LIN {X 0,Y 236.582,Z 268.091,A -85,B 0,C 180,E1 -19847.962,E2 -19847.962} C_VEL
LIN {X 0,Y 237.174,Z 271.955,A -85,B 0,C 180,E1 -19851.515,E2 -19851.515} C_VEL
LIN {X 0,Y 237.168,Z 273.271,A -85,B 0,C 180,E1 -19852.68,E2 -19852.68} C_VEL
LIN {X 0,Y 236.828,Z 274.344,A -85,B 0,C 180,E1 -19853.588,E2 -19853.588} C_VEL
LIN {X 0,Y 235.899,Z 275.46,A -85,B 0,C 180,E1 -19854.474,E2 -19854.474} C_VEL
LIN {X 0,Y 233.05,Z 277.73,A -85,B 0,C 180,E1 -19856.2,E2 -19856.2} C_VEL
LIN {X 0,Y 230.018,Z 280.043,A -85,B 0,C 180,E1 -19857.965,E2 -19857.965} C_VEL
LIN {X 0,Y 228.529,Z 281.776,A -85,B 0,C 180,E1 -19859.356,E2 -19859.356} C_VEL
LIN {X 0,Y 228.311,Z 282.347,A -85,B 0,C 180,E1 -19859.835,E2 -19859.835} C_VEL
LIN {X 0,Y 228.093,Z 283.329,A -85,B 0,C 180,E1 -19860.667,E2 -19860.667} C_VEL
LIN {X 0,Y 230.544,Z 296.949,A -85,B 0,C 180,E1 -19861.77,E2 -19861.77} C_VEL
LIN {X 0,Y 232.298,Z 310.068,A -85,B 0,C 180,E1 -19863.141,E2 -19863.141} C_VEL
LIN {X 0,Y 233.32,Z 321.823,A -85,B 0,C 180,E1 -19864.647,E2 -19864.647} C_VEL
LIN {X 0,Y 233.838,Z 332.507,A -85,B 0,C 180,E1 -19866.296,E2 -19866.296} C_VEL
LIN {X 0,Y 233.74,Z 339.045,A -85,B 0,C 180,E1 -19867.456,E2 -19867.456} C_VEL
LIN {X 0,Y 231.671,Z 349.675,A -85,B 0,C 180,E1 -19869.58,E2 -19869.58} C_VEL
LIN {X 0,Y 229.872,Z 358.64,A -85,B 0,C 180,E1 -19871.823,E2 -19871.823} C_VEL
LIN {X 0,Y 228.341,Z 366.767,A -85,B 0,C 180,E1 -19874.375,E2 -19874.375} C_VEL
LIN {X 0,Y 227.062,Z 373.529,A -85,B 0,C 180,E1 -19877.031,E2 -19877.031} C_VEL
LIN {X 0,Y 226.239,Z 379.732,A -85,B 0,C 180,E1 -19880.161,E2 -19880.161} C_VEL
LIN {X 0,Y 225.922,Z 383.732,A -85,B 0,C 180,E1 -19882.85,E2 -19882.85} C_VEL
LIN {X 0,Y 225.93,Z 385.778,A -85,B 0,C 180,E1 -19884.644,E2 -19884.644} C_VEL
LIN {X 0,Y 225.893,Z 387.38,A -85,B 0,C 180,E1 -19886.431,E2 -19886.431} C_VEL
LIN {X 0,Y 225.931,Z 388.566,A -85,B 0,C 180,E1 -19888.216,E2 -19888.216} C_VEL
LIN {X 0,Y 225.973,Z 389.31,A -85,B 0,C 180,E1 -19889.998,E2 -19889.998} C_VEL
LIN {X 0,Y 225.893,Z 389.616,A -85,B 0,C 180,E1 -19891.781,E2 -19891.781} C_VEL
LIN {X 0,Y 225.727,Z 389.197,A -85,B 0,C 180,E1 -19894.896,E2 -19894.896} C_VEL
LIN {X 0,Y 225.828,Z 388.167,A -85,B 0,C 180,E1 -19897.149,E2 -19897.149} C_VEL
LIN {X 0,Y 226.44,Z 385.148,A -85,B 0,C 180,E1 -19900.731,E2 -19900.731} C_VEL
LIN {X 0,Y 227.36,Z 381.799,A -85,B 0,C 180,E1 -19903.403,E2 -19903.403} C_VEL
LIN {X 0,Y 228.933,Z 377.423,A -85,B 0,C 180,E1 -19906.037,E2 -19906.037} C_VEL
LIN {X 0,Y 231.289,Z 370.883,A -85,B 0,C 180,E1 -19909.064,E2 -19909.064} C_VEL
LIN {X 0,Y 233.668,Z 363.826,A -85,B 0,C 180,E1 -19911.618,E2 -19911.618} C_VEL
LIN {X 0,Y 236.692,Z 355.088,A -85,B 0,C 180,E1 -19914.094,E2 -19914.094} C_VEL
LIN {X 0,Y 239.624,Z 346.258,A -85,B 0,C 180,E1 -19916.098,E2 -19916.098} C_VEL
LIN {X 0,Y 240.747,Z 338.01,A -85,B 0,C 180,E1 -19917.843,E2 -19917.843} C_VEL
LIN {X 0,Y 241.168,Z 328.351,A -85,B 0,C 180,E1 -19919.694,E2 -19919.694} C_VEL
LIN {X 0,Y 240.657,Z 317.965,A -85,B 0,C 180,E1 -19921.527,E2 -19921.527} C_VEL
LIN {X 0,Y 239.299,Z 308.276,A -85,B 0,C 180,E1 -19923.171,E2 -19923.171} C_VEL
LIN {X 0,Y 236.551,Z 295.925,A -85,B 0,C 180,E1 -19925.187,E2 -19925.187} C_VEL
LIN {X 0,Y 233.987,Z 287.833,A -85,B 0,C 180,E1 -19926.545,E2 -19926.545} C_VEL
LIN {X 0,Y 232.504,Z 283.742,A -85,B 0,C 180,E1 -19927.235,E2 -19927.235} C_VEL
LIN {X 0,Y 231.232,Z 280.621,A -85,B 0,C 180,E1 -19927.789,E2 -19927.789} C_VEL
LIN {X 0,Y 231.06,Z 279.554,A -85,B 0,C 180,E1 -19927.942,E2 -19927.942} C_VEL
LIN {X 0,Y 230.865,Z 277.251,A -85,B 0,C 180,E1 -19930.44,E2 -19930.44} C_VEL
LIN {X 0,Y 230.241,Z 273.767,A -85,B 0,C 180,E1 -19934.59,E2 -19934.59} C_VEL
LIN {X 0,Y 229.813,Z 271.38,A -85,B 0,C 180,E1 -19937.714,E2 -19937.714} C_VEL
LIN {X 0,Y 229.314,Z 268.321,A -85,B 0,C 180,E1 -19942.193,E2 -19942.193} C_VEL
LIN {X 0,Y 228.917,Z 265.854,A -85,B 0,C 180,E1 -19946.45,E2 -19946.45} C_VEL
LIN {X 0,Y 228.589,Z 263.894,A -85,B 0,C 180,E1 -19950.53,E2 -19950.53} C_VEL
LIN {X 0,Y 228.326,Z 262.331,A -85,B 0,C 180,E1 -19954.471,E2 -19954.471} C_VEL
LIN {X 0,Y 228.146,Z 261.159,A -85,B 0,C 180,E1 -19958.303,E2 -19958.303} C_VEL
LIN {X 0,Y 228.044,Z 260.181,A -85,B 0,C 180,E1 -19962.812,E2 -19962.812} C_VEL
LIN {X 0,Y 228.091,Z 260.073,A -85,B 0,C 180,E1 -19967.542,E2 -19967.542} C_VEL
LIN {X 0,Y 228.321,Z 260.045,A -85,B 0,C 180,E1 -19971.144,E2 -19971.144} C_VEL
LIN {X 0,Y 228.353,Z 260.04,A -85,B 0,C 180,E1 -19972.926,E2 -19972.926} C_VEL
LIN {X 0,Y 228.55,Z 260.016,A -85,B 0,C 180,E1 -19978.235,E2 -19978.235} C_VEL
LIN {X 0,Y 228.611,Z 260.556,A -85,B 0,C 180,E1 -19981.759,E2 -19981.759} C_VEL
LIN {X 0,Y 228.635,Z 261.873,A -85,B 0,C 180,E1 -19987.06,E2 -19987.06} C_VEL
LIN {X 0,Y 228.673,Z 262.986,A -85,B 0,C 180,E1 -19990.623,E2 -19990.623} C_VEL
LIN {X 0,Y 228.643,Z 264.459,A -85,B 0,C 180,E1 -19994.573,E2 -19994.573} C_VEL
LIN {X 0,Y 229.76,Z 267.333,A -85,B 0,C 180,E1 -19995.124,E2 -19995.124} C_VEL
LIN {X 0,Y 231.658,Z 269.874,A -85,B 0,C 180,E1 -19995.842,E2 -19995.842} C_VEL
LIN {X 0,Y 233.644,Z 273.431,A -85,B 0,C 180,E1 -19996.696,E2 -19996.696} C_VEL
LIN {X 0,Y 237.42,Z 281.431,A -85,B 0,C 180,E1 -19998.483,E2 -19998.483} C_VEL
LIN {X 0,Y 240.96,Z 290.866,A -85,B 0,C 180,E1 -20000.484,E2 -20000.484} C_VEL
LIN {X 0,Y 243.397,Z 299.783,A -85,B 0,C 180,E1 -20002.367,E2 -20002.367} C_VEL
LIN {X 0,Y 245.117,Z 310.056,A -85,B 0,C 180,E1 -20004.563,E2 -20004.563} C_VEL
LIN {X 0,Y 245.334,Z 313.056,A -85,B 0,C 180,E1 -20005.218,E2 -20005.218} C_VEL
LIN {X 0,Y 242.951,Z 322.016,A -85,B 0,C 180,E1 -20006.862,E2 -20006.862} C_VEL
LIN {X 0,Y 240.35,Z 330.299,A -85,B 0,C 180,E1 -20008.695,E2 -20008.695} C_VEL
LIN {X 0,Y 237.533,Z 338.398,A -85,B 0,C 180,E1 -20010.907,E2 -20010.907} C_VEL
LIN {X 0,Y 234.499,Z 346.25,A -85,B 0,C 180,E1 -20013.621,E2 -20013.621} C_VEL
LIN {X 0,Y 231.903,Z 352.66,A -85,B 0,C 180,E1 -20016.5,E2 -20016.5} C_VEL
LIN {X 0,Y 230.178,Z 356.698,A -85,B 0,C 180,E1 -20018.873,E2 -20018.873} C_VEL
LIN {X 0,Y 228.237,Z 360.993,A -85,B 0,C 180,E1 -20022.355,E2 -20022.355} C_VEL
LIN {X 0,Y 226.997,Z 363.354,A -85,B 0,C 180,E1 -20025.401,E2 -20025.401} C_VEL
LIN {X 0,Y 226.239,Z 364.471,A -85,B 0,C 180,E1 -20028.201,E2 -20028.201} C_VEL
LIN {X 0,Y 225.758,Z 364.552,A -85,B 0,C 180,E1 -20031.495,E2 -20031.495} C_VEL
LIN {X 0,Y 225.655,Z 363.668,A -85,B 0,C 180,E1 -20034.067,E2 -20034.067} C_VEL
LIN {X 0,Y 225.915,Z 361.541,A -85,B 0,C 180,E1 -20037.128,E2 -20037.128} C_VEL
LIN {X 0,Y 226.555,Z 358.042,A -85,B 0,C 180,E1 -20040.289,E2 -20040.289} C_VEL
LIN {X 0,Y 227.494,Z 352.709,A -85,B 0,C 180,E1 -20043.616,E2 -20043.616} C_VEL
LIN {X 0,Y 228.704,Z 346.677,A -85,B 0,C 180,E1 -20046.456,E2 -20046.456} C_VEL
LIN {X 0,Y 230.139,Z 339.915,A -85,B 0,C 180,E1 -20048.974,E2 -20048.974} C_VEL
LIN {X 0,Y 231.82,Z 331.64,A -85,B 0,C 180,E1 -20051.44,E2 -20051.44} C_VEL
LIN {X 0,Y 233.769,Z 322.282,A -85,B 0,C 180,E1 -20053.677,E2 -20053.677} C_VEL
LIN {X 0,Y 235.788,Z 311.376,A -85,B 0,C 180,E1 -20055.767,E2 -20055.767} C_VEL
LIN {X 0,Y 237.189,Z 302.379,A -85,B 0,C 180,E1 -20057.162,E2 -20057.162} C_VEL
LIN {X 0,Y 235.414,Z 291.626,A -85,B 0,C 180,E1 -20058.813,E2 -20058.813} C_VEL
LIN {X 0,Y 232.759,Z 279.44,A -85,B 0,C 180,E1 -20060.4,E2 -20060.4} C_VEL
LIN {X 0,Y 229.192,Z 266.831,A -85,B 0,C 180,E1 -20061.788,E2 -20061.788} C_VEL
LIN {X 0,Y 227.359,Z 260.437,A -85,B 0,C 180,E1 -20062.392,E2 -20062.392} C_VEL
LIN {X 0,Y 227.394,Z 260.162,A -85,B 0,C 180,E1 -20062.9,E2 -20062.9} C_VEL
LIN {X 0,Y 227.807,Z 260.108,A -85,B 0,C 180,E1 -20066.464,E2 -20066.464} C_VEL
LIN {X 0,Y 228.552,Z 260.014,A -85,B 0,C 180,E1 -20070.002,E2 -20070.002} C_VEL
LIN {X 0,Y 228.543,Z 260.017,A -85,B 0,C 180,E1 -20071.764,E2 -20071.764} C_VEL
LIN {X 0,Y 228.343,Z 260.043,A -85,B 0,C 180,E1 -20077.074,E2 -20077.074} C_VEL
LIN {X 0,Y 228.152,Z 260.064,A -85,B 0,C 180,E1 -20080.653,E2 -20080.653} C_VEL
LIN {X 0,Y 228.055,Z 260.077,A -85,B 0,C 180,E1 -20086.104,E2 -20086.104} C_VEL
LIN {X 0,Y 227.955,Z 260.089,A -85,B 0,C 180,E1 -20089.826,E2 -20089.826} C_VEL
LIN {X 0,Y 227.92,Z 260.094,A -85,B 0,C 180,E1 -20093.634,E2 -20093.634} C_VEL
LIN {X 0,Y 227.878,Z 260.1,A -85,B 0,C 180,E1 -20097.558,E2 -20097.558} C_VEL
LIN {X 0,Y 227.866,Z 260.102,A -85,B 0,C 180,E1 -20101.625,E2 -20101.625} C_VEL
LIN {X 0,Y 227.895,Z 260.097,A -85,B 0,C 180,E1 -20105.871,E2 -20105.871} C_VEL
LIN {X 0,Y 227.887,Z 260.097,A -85,B 0,C 180,E1 -20110.366,E2 -20110.366} C_VEL
LIN {X 0,Y 227.905,Z 260.097,A -85,B 0,C 180,E1 -20112.723,E2 -20112.723} C_VEL
LIN {X 0,Y 227.895,Z 260.095,A -85,B 0,C 180,E1 -20117.745,E2 -20117.745} C_VEL
LIN {X 0,Y 227.869,Z 260.097,A -85,B 0,C 180,E1 -20121.918,E2 -20121.918} C_VEL
LIN {X 0,Y 227.889,Z 260.084,A -85,B 0,C 180,E1 -20126.377,E2 -20126.377} C_VEL
LIN {X 0,Y 227.918,Z 260.094,A -85,B 0,C 180,E1 -20130.441,E2 -20130.441} C_VEL
LIN {X 0,Y 227.93,Z 260.091,A -85,B 0,C 180,E1 -20134.429,E2 -20134.429} C_VEL
LIN {X 0,Y 227.965,Z 260.076,A -85,B 0,C 180,E1 -20138.291,E2 -20138.291} C_VEL
LIN {X 0,Y 228.039,Z 260.072,A -85,B 0,C 180,E1 -20142.829,E2 -20142.829} C_VEL
LIN {X 0,Y 228.097,Z 260.071,A -85,B 0,C 180,E1 -20147.548,E2 -20147.548} C_VEL
LIN {X 0,Y 228.269,Z 260.044,A -85,B 0,C 180,E1 -20151.147,E2 -20151.147} C_VEL
LIN {X 0,Y 228.324,Z 260.031,A -85,B 0,C 180,E1 -20152.93,E2 -20152.93} C_VEL
LIN {X 0,Y 228.56,Z 260.012,A -85,B 0,C 180,E1 -20158.241,E2 -20158.241} C_VEL
LIN {X 0,Y 228.56,Z 260.016,A -85,B 0,C 180,E1 -20161.765,E2 -20161.765} C_VEL
LIN {X 0,Y 228.322,Z 260.033,A -85,B 0,C 180,E1 -20167.075,E2 -20167.075} C_VEL
LIN {X 0,Y 228.154,Z 260.06,A -85,B 0,C 180,E1 -20170.653,E2 -20170.653} C_VEL
LIN {X 0,Y 228.072,Z 260.074,A -85,B 0,C 180,E1 -20174.274,E2 -20174.274} C_VEL
LIN {X 0,Y 228.014,Z 260.073,A -85,B 0,C 180,E1 -20177.955,E2 -20177.955} C_VEL
LIN {X 0,Y 227.941,Z 260.09,A -85,B 0,C 180,E1 -20182.331,E2 -20182.331} C_VEL
LIN {X 0,Y 227.953,Z 260.086,A -85,B 0,C 180,E1 -20186.604,E2 -20186.604} C_VEL
LIN {X 0,Y 227.908,Z 260.094,A -85,B 0,C 180,E1 -20190.292,E2 -20190.292} C_VEL
LIN {X 0,Y 227.888,Z 260.097,A -85,B 0,C 180,E1 -20193.721,E2 -20193.721} C_VEL
LIN {X 0,Y 227.932,Z 260.16,A -85,B 0,C 180,E1 -20198.668,E2 -20198.668} C_VEL
LIN {X 0,Y 228.56,Z 263.745,A -85,B 0,C 180,E1 -20202.572,E2 -20202.572} C_VEL
LIN {X 0,Y 229.474,Z 268.735,A -85,B 0,C 180,E1 -20207.638,E2 -20207.638} C_VEL
LIN {X 0,Y 230.081,Z 272.478,A -85,B 0,C 180,E1 -20211.228,E2 -20211.228} C_VEL
LIN {X 0,Y 230.054,Z 275.028,A -85,B 0,C 180,E1 -20213.546,E2 -20213.546} C_VEL
LIN {X 0,Y 228.962,Z 279.607,A -85,B 0,C 180,E1 -20217.507,E2 -20217.507} C_VEL
LIN {X 0,Y 228.311,Z 282.347,A -85,B 0,C 180,E1 -20219.835,E2 -20219.835} C_VEL
LIN {X 0,Y 228.247,Z 283.713,A -85,B 0,C 180,E1 -20220.368,E2 -20220.368} C_VEL
LIN {X 0,Y 228.252,Z 286.665,A -85,B 0,C 180,E1 -20220.831,E2 -20220.831} C_VEL
LIN {X 0,Y 227.557,Z 295.044,A -85,B 0,C 180,E1 -20221.333,E2 -20221.333} C_VEL
LIN {X 0,Y 225.695,Z 307.555,A -85,B 0,C 180,E1 -20222.229,E2 -20222.229} C_VEL
LIN {X 0,Y 225.598,Z 311.732,A -85,B 0,C 180,E1 -20222.718,E2 -20222.718} C_VEL
LIN {X 0,Y 226.563,Z 323.939,A -85,B 0,C 180,E1 -20224.408,E2 -20224.408} C_VEL
LIN {X 0,Y 226.931,Z 334.996,A -85,B 0,C 180,E1 -20226.257,E2 -20226.257} C_VEL
LIN {X 0,Y 226.737,Z 340.013,A -85,B 0,C 180,E1 -20227.202,E2 -20227.202} C_VEL
LIN {X 0,Y 224.973,Z 348.459,A -85,B 0,C 180,E1 -20228.944,E2 -20228.944} C_VEL
LIN {X 0,Y 223.066,Z 357.154,A -85,B 0,C 180,E1 -20231.131,E2 -20231.131} C_VEL
LIN {X 0,Y 221.983,Z 363.183,A -85,B 0,C 180,E1 -20232.969,E2 -20232.969} C_VEL
LIN {X 0,Y 220.543,Z 370.59,A -85,B 0,C 180,E1 -20235.7,E2 -20235.7} C_VEL
LIN {X 0,Y 219.632,Z 375.607,A -85,B 0,C 180,E1 -20237.993,E2 -20237.993} C_VEL
LIN {X 0,Y 219.049,Z 380.469,A -85,B 0,C 180,E1 -20240.767,E2 -20240.767} C_VEL
LIN {X 0,Y 218.844,Z 384.179,A -85,B 0,C 180,E1 -20243.544,E2 -20243.544} C_VEL
LIN {X 0,Y 218.815,Z 386.828,A -85,B 0,C 180,E1 -20246.315,E2 -20246.315} C_VEL
LIN {X 0,Y 218.861,Z 388.048,A -85,B 0,C 180,E1 -20248.158,E2 -20248.158} C_VEL
LIN {X 0,Y 218.899,Z 388.852,A -85,B 0,C 180,E1 -20249.998,E2 -20249.998} C_VEL
LIN {X 0,Y 218.819,Z 389.197,A -85,B 0,C 180,E1 -20251.839,E2 -20251.839} C_VEL
LIN {X 0,Y 218.658,Z 388.69,A -85,B 0,C 180,E1 -20255.531,E2 -20255.531} C_VEL
LIN {X 0,Y 218.757,Z 387.862,A -85,B 0,C 180,E1 -20257.381,E2 -20257.381} C_VEL
LIN {X 0,Y 218.998,Z 386.61,A -85,B 0,C 180,E1 -20259.232,E2 -20259.232} C_VEL
LIN {X 0,Y 220.005,Z 382.872,A -85,B 0,C 180,E1 -20262.919,E2 -20262.919} C_VEL
LIN {X 0,Y 221.485,Z 378.926,A -85,B 0,C 180,E1 -20265.645,E2 -20265.645} C_VEL
LIN {X 0,Y 223.37,Z 373.893,A -85,B 0,C 180,E1 -20268.337,E2 -20268.337} C_VEL
LIN {X 0,Y 225.873,Z 367.269,A -85,B 0,C 180,E1 -20271.124,E2 -20271.124} C_VEL
LIN {X 0,Y 228.568,Z 359.988,A -85,B 0,C 180,E1 -20273.559,E2 -20273.559} C_VEL
LIN {X 0,Y 232.041,Z 350.477,A -85,B 0,C 180,E1 -20276.049,E2 -20276.049} C_VEL
LIN {X 0,Y 233.674,Z 344.927,A -85,B 0,C 180,E1 -20277.299,E2 -20277.299} C_VEL
LIN {X 0,Y 234.841,Z 334.364,A -85,B 0,C 180,E1 -20279.568,E2 -20279.568} C_VEL
LIN {X 0,Y 234.903,Z 324.058,A -85,B 0,C 180,E1 -20281.578,E2 -20281.578} C_VEL
LIN {X 0,Y 233.981,Z 313.378,A -85,B 0,C 180,E1 -20283.535,E2 -20283.535} C_VEL
LIN {X 0,Y 231.901,Z 302.017,A -85,B 0,C 180,E1 -20285.546,E2 -20285.546} C_VEL
LIN {X 0,Y 229.361,Z 292.372,A -85,B 0,C 180,E1 -20287.273,E2 -20287.273} C_VEL
LIN {X 0,Y 227.435,Z 286.944,A -85,B 0,C 180,E1 -20288.297,E2 -20288.297} C_VEL
LIN {X 0,Y 226.256,Z 284.042,A -85,B 0,C 180,E1 -20288.857,E2 -20288.857} C_VEL
LIN {X 0,Y 224.405,Z 280.75,A -85,B 0,C 180,E1 -20289.658,E2 -20289.658} C_VEL
LIN {X 0,Y 223.937,Z 278.935,A -85,B 0,C 180,E1 -20289.96,E2 -20289.96} C_VEL
LIN {X 0,Y 223.376,Z 275.767,A -85,B 0,C 180,E1 -20293.8,E2 -20293.8} C_VEL
LIN {X 0,Y 222.755,Z 272.287,A -85,B 0,C 180,E1 -20298.502,E2 -20298.502} C_VEL
LIN {X 0,Y 222.291,Z 269.349,A -85,B 0,C 180,E1 -20303.076,E2 -20303.076} C_VEL
LIN {X 0,Y 221.88,Z 267.008,A -85,B 0,C 180,E1 -20307.418,E2 -20307.418} C_VEL
LIN {X 0,Y 221.586,Z 265.096,A -85,B 0,C 180,E1 -20311.589,E2 -20311.589} C_VEL
LIN {X 0,Y 221.346,Z 263.637,A -85,B 0,C 180,E1 -20315.619,E2 -20315.619} C_VEL
LIN {X 0,Y 221.178,Z 262.571,A -85,B 0,C 180,E1 -20319.539,E2 -20319.539} C_VEL
LIN {X 0,Y 221.152,Z 261.793,A -85,B 0,C 180,E1 -20323.378,E2 -20323.378} C_VEL
LIN {X 0,Y 221.144,Z 261.239,A -85,B 0,C 180,E1 -20329.005,E2 -20329.005} C_VEL
LIN {X 0,Y 221.328,Z 261.175,A -85,B 0,C 180,E1 -20332.7,E2 -20332.7} C_VEL
LIN {X 0,Y 221.614,Z 261.562,A -85,B 0,C 180,E1 -20338.18,E2 -20338.18} C_VEL
LIN {X 0,Y 221.745,Z 261.799,A -85,B 0,C 180,E1 -20339.997,E2 -20339.997} C_VEL
LIN {X 0,Y 221.511,Z 262.564,A -85,B 0,C 180,E1 -20343.635,E2 -20343.635} C_VEL
LIN {X 0,Y 221.7,Z 263.426,A -85,B 0,C 180,E1 -20347.282,E2 -20347.282} C_VEL
LIN {X 0,Y 221.655,Z 264.878,A -85,B 0,C 180,E1 -20351.891,E2 -20351.891} C_VEL
LIN {X 0,Y 221.7,Z 265.259,A -85,B 0,C 180,E1 -20352.527,E2 -20352.527} C_VEL
LIN {X 0,Y 222.844,Z 268.053,A -85,B 0,C 180,E1 -20353.135,E2 -20353.135} C_VEL
LIN {X 0,Y 224.868,Z 270.638,A -85,B 0,C 180,E1 -20353.989,E2 -20353.989} C_VEL
LIN {X 0,Y 226.934,Z 274.226,A -85,B 0,C 180,E1 -20354.972,E2 -20354.972} C_VEL
LIN {X 0,Y 231.406,Z 283.228,A -85,B 0,C 180,E1 -20357.221,E2 -20357.221} C_VEL
LIN {X 0,Y 234.702,Z 291.81,A -85,B 0,C 180,E1 -20359.229,E2 -20359.229} C_VEL
LIN {X 0,Y 237.218,Z 300.932,A -85,B 0,C 180,E1 -20361.277,E2 -20361.277} C_VEL
LIN {X 0,Y 238.783,Z 310.302,A -85,B 0,C 180,E1 -20363.414,E2 -20363.414} C_VEL
LIN {X 0,Y 239.148,Z 314.984,A -85,B 0,C 180,E1 -20364.499,E2 -20364.499} C_VEL
LIN {X 0,Y 235.909,Z 325.925,A -85,B 0,C 180,E1 -20366.658,E2 -20366.658} C_VEL
LIN {X 0,Y 232.762,Z 334.933,A -85,B 0,C 180,E1 -20368.885,E2 -20368.885} C_VEL
LIN {X 0,Y 229.807,Z 342.679,A -85,B 0,C 180,E1 -20371.322,E2 -20371.322} C_VEL
LIN {X 0,Y 226.581,Z 350.194,A -85,B 0,C 180,E1 -20374.345,E2 -20374.345} C_VEL
LIN {X 0,Y 224.11,Z 355.72,A -85,B 0,C 180,E1 -20377.304,E2 -20377.304} C_VEL
LIN {X 0,Y 222.062,Z 360.132,A -85,B 0,C 180,E1 -20380.577,E2 -20380.577} C_VEL
LIN {X 0,Y 220.85,Z 362.435,A -85,B 0,C 180,E1 -20382.955,E2 -20382.955} C_VEL
LIN {X 0,Y 219.917,Z 363.987,A -85,B 0,C 180,E1 -20385.329,E2 -20385.329} C_VEL
LIN {X 0,Y 219.263,Z 364.857,A -85,B 0,C 180,E1 -20387.695,E2 -20387.695} C_VEL
LIN {X 0,Y 218.757,Z 365.07,A -85,B 0,C 180,E1 -20390.443,E2 -20390.443} C_VEL
LIN {X 0,Y 218.581,Z 364.271,A -85,B 0,C 180,E1 -20393.491,E2 -20393.491} C_VEL
LIN {X 0,Y 218.781,Z 362.082,A -85,B 0,C 180,E1 -20396.903,E2 -20396.903} C_VEL
LIN {X 0,Y 219.367,Z 358.998,A -85,B 0,C 180,E1 -20399.877,E2 -20399.877} C_VEL
LIN {X 0,Y 220.269,Z 353.967,A -85,B 0,C 180,E1 -20403.293,E2 -20403.293} C_VEL
LIN {X 0,Y 221.481,Z 348.036,A -85,B 0,C 180,E1 -20406.272,E2 -20406.272} C_VEL
LIN {X 0,Y 223.163,Z 340.423,A -85,B 0,C 180,E1 -20409.252,E2 -20409.252} C_VEL
LIN {X 0,Y 224.875,Z 332.191,A -85,B 0,C 180,E1 -20411.79,E2 -20411.79} C_VEL
LIN {X 0,Y 226.732,Z 323.661,A -85,B 0,C 180,E1 -20413.913,E2 -20413.913} C_VEL
LIN {X 0,Y 228.736,Z 313.328,A -85,B 0,C 180,E1 -20416,E2 -20416} C_VEL
LIN {X 0,Y 230.335,Z 303.125,A -85,B 0,C 180,E1 -20417.669,E2 -20417.669} C_VEL
LIN {X 0,Y 228.601,Z 292.522,A -85,B 0,C 180,E1 -20419.372,E2 -20419.372} C_VEL
LIN {X 0,Y 226.174,Z 281.326,A -85,B 0,C 180,E1 -20420.899,E2 -20420.899} C_VEL
LIN {X 0,Y 222.52,Z 268.016,A -85,B 0,C 180,E1 -20422.433,E2 -20422.433} C_VEL
LIN {X 0,Y 220.395,Z 261.032,A -85,B 0,C 180,E1 -20423.134,E2 -20423.134} C_VEL
LIN {X 0,Y 221.15,Z 260.936,A -85,B 0,C 180,E1 -20428.181,E2 -20428.181} C_VEL
LIN {X 0,Y 221.511,Z 260.891,A -85,B 0,C 180,E1 -20430.002,E2 -20430.002} C_VEL
LIN {X 0,Y 221.501,Z 260.894,A -85,B 0,C 180,E1 -20431.82,E2 -20431.82} C_VEL
LIN {X 0,Y 221.278,Z 260.922,A -85,B 0,C 180,E1 -20437.301,E2 -20437.301} C_VEL
LIN {X 0,Y 221.101,Z 260.944,A -85,B 0,C 180,E1 -20440.997,E2 -20440.997} C_VEL
LIN {X 0,Y 221.015,Z 260.955,A -85,B 0,C 180,E1 -20446.632,E2 -20446.632} C_VEL
LIN {X 0,Y 220.911,Z 260.968,A -85,B 0,C 180,E1 -20450.486,E2 -20450.486} C_VEL
LIN {X 0,Y 220.866,Z 260.974,A -85,B 0,C 180,E1 -20454.437,E2 -20454.437} C_VEL
LIN {X 0,Y 220.829,Z 260.98,A -85,B 0,C 180,E1 -20458.517,E2 -20458.517} C_VEL
LIN {X 0,Y 220.817,Z 260.981,A -85,B 0,C 180,E1 -20462.758,E2 -20462.758} C_VEL
LIN {X 0,Y 220.833,Z 260.977,A -85,B 0,C 180,E1 -20467.291,E2 -20467.291} C_VEL
LIN {X 0,Y 220.849,Z 260.974,A -85,B 0,C 180,E1 -20471.936,E2 -20471.936} C_VEL
LIN {X 0,Y 220.858,Z 260.973,A -85,B 0,C 180,E1 -20477.048,E2 -20477.048} C_VEL
LIN {X 0,Y 220.849,Z 260.974,A -85,B 0,C 180,E1 -20480.477,E2 -20480.477} C_VEL
LIN {X 0,Y 220.814,Z 260.961,A -85,B 0,C 180,E1 -20485.052,E2 -20485.052} C_VEL
LIN {X 0,Y 220.868,Z 260.967,A -85,B 0,C 180,E1 -20489.399,E2 -20489.399} C_VEL
LIN {X 0,Y 220.896,Z 260.967,A -85,B 0,C 180,E1 -20493.553,E2 -20493.553} C_VEL
LIN {X 0,Y 220.88,Z 260.962,A -85,B 0,C 180,E1 -20497.557,E2 -20497.557} C_VEL
LIN {X 0,Y 220.988,Z 260.951,A -85,B 0,C 180,E1 -20502.575,E2 -20502.575} C_VEL
LIN {X 0,Y 221.03,Z 260.95,A -85,B 0,C 180,E1 -20507.143,E2 -20507.143} C_VEL
LIN {X 0,Y 221.207,Z 260.923,A -85,B 0,C 180,E1 -20510.862,E2 -20510.862} C_VEL
LIN {X 0,Y 221.26,Z 260.911,A -85,B 0,C 180,E1 -20512.704,E2 -20512.704} C_VEL
LIN {X 0,Y 221.518,Z 260.889,A -85,B 0,C 180,E1 -20518.185,E2 -20518.185} C_VEL
LIN {X 0,Y 221.517,Z 260.893,A -85,B 0,C 180,E1 -20521.821,E2 -20521.821} C_VEL
LIN {X 0,Y 221.258,Z 260.912,A -85,B 0,C 180,E1 -20527.302,E2 -20527.302} C_VEL
LIN {X 0,Y 221.075,Z 260.943,A -85,B 0,C 180,E1 -20530.999,E2 -20530.999} C_VEL
LIN {X 0,Y 221.027,Z 260.949,A -85,B 0,C 180,E1 -20536.632,E2 -20536.632} C_VEL
LIN {X 0,Y 220.903,Z 260.963,A -85,B 0,C 180,E1 -20540.488,E2 -20540.488} C_VEL
LIN {X 0,Y 220.878,Z 260.97,A -85,B 0,C 180,E1 -20544.436,E2 -20544.436} C_VEL
LIN {X 0,Y 220.838,Z 260.97,A -85,B 0,C 180,E1 -20548.516,E2 -20548.516} C_VEL
LIN {X 0,Y 220.827,Z 260.978,A -85,B 0,C 180,E1 -20552.757,E2 -20552.757} C_VEL
LIN {X 0,Y 220.849,Z 260.974,A -85,B 0,C 180,E1 -20557.779,E2 -20557.779} C_VEL
LIN {X 0,Y 220.856,Z 261.088,A -85,B 0,C 180,E1 -20558.356,E2 -20558.356} C_VEL
LIN {X 0,Y 221.422,Z 264.152,A -85,B 0,C 180,E1 -20561.804,E2 -20561.804} C_VEL
LIN {X 0,Y 222.239,Z 268.736,A -85,B 0,C 180,E1 -20566.667,E2 -20566.667} C_VEL
LIN {X 0,Y 222.999,Z 273.012,A -85,B 0,C 180,E1 -20570.924,E2 -20570.924} C_VEL
LIN {X 0,Y 223.009,Z 275.438,A -85,B 0,C 180,E1 -20573.216,E2 -20573.216} C_VEL
LIN {X 0,Y 222.507,Z 277.787,A -85,B 0,C 180,E1 -20575.349,E2 -20575.349} C_VEL
LIN {X 0,Y 221.196,Z 282.96,A -85,B 0,C 180,E1 -20579.905,E2 -20579.905} C_VEL
LIN {X 0,Y 223.81,Z 297.497,A -85,B 0,C 180,E1 -20581.15,E2 -20581.15} C_VEL
LIN {X 0,Y 225.422,Z 310.201,A -85,B 0,C 180,E1 -20582.532,E2 -20582.532} C_VEL
LIN {X 0,Y 225.598,Z 311.732,A -85,B 0,C 180,E1 -20582.718,E2 -20582.718} C_VEL
LIN {X 0,Y 225.445,Z 317.098,A -85,B 0,C 180,E1 -20583.36,E2 -20583.36} C_VEL
LIN {X 0,Y 223.352,Z 325.814,A -85,B 0,C 180,E1 -20584.431,E2 -20584.431} C_VEL
LIN {X 0,Y 221.242,Z 332.584,A -85,B 0,C 180,E1 -20585.395,E2 -20585.395} C_VEL
LIN {X 0,Y 219.95,Z 339.014,A -85,B 0,C 180,E1 -20586.543,E2 -20586.543} C_VEL
LIN {X 0,Y 218.294,Z 347.241,A -85,B 0,C 180,E1 -20588.267,E2 -20588.267} C_VEL
LIN {X 0,Y 216.457,Z 355.711,A -85,B 0,C 180,E1 -20590.42,E2 -20590.42} C_VEL
LIN {X 0,Y 214.836,Z 363.567,A -85,B 0,C 180,E1 -20592.875,E2 -20592.875} C_VEL
LIN {X 0,Y 213.384,Z 370.834,A -85,B 0,C 180,E1 -20595.697,E2 -20595.697} C_VEL
LIN {X 0,Y 212.38,Z 376.628,A -85,B 0,C 180,E1 -20598.546,E2 -20598.546} C_VEL
LIN {X 0,Y 211.875,Z 381.169,A -85,B 0,C 180,E1 -20601.414,E2 -20601.414} C_VEL
LIN {X 0,Y 211.801,Z 384.857,A -85,B 0,C 180,E1 -20604.563,E2 -20604.563} C_VEL
LIN {X 0,Y 211.791,Z 387.524,A -85,B 0,C 180,E1 -20608.096,E2 -20608.096} C_VEL
LIN {X 0,Y 211.828,Z 388.366,A -85,B 0,C 180,E1 -20609.998,E2 -20609.998} C_VEL
LIN {X 0,Y 211.745,Z 388.775,A -85,B 0,C 180,E1 -20611.9,E2 -20611.9} C_VEL
LIN {X 0,Y 211.576,Z 388.339,A -85,B 0,C 180,E1 -20615.717,E2 -20615.717} C_VEL
LIN {X 0,Y 211.944,Z 386.362,A -85,B 0,C 180,E1 -20619.542,E2 -20619.542} C_VEL
LIN {X 0,Y 213.05,Z 382.706,A -85,B 0,C 180,E1 -20623.349,E2 -20623.349} C_VEL
LIN {X 0,Y 214.631,Z 378.851,A -85,B 0,C 180,E1 -20626.158,E2 -20626.158} C_VEL
LIN {X 0,Y 216.632,Z 373.93,A -85,B 0,C 180,E1 -20628.928,E2 -20628.928} C_VEL
LIN {X 0,Y 219.134,Z 367.697,A -85,B 0,C 180,E1 -20631.689,E2 -20631.689} C_VEL
LIN {X 0,Y 222.081,Z 360.273,A -85,B 0,C 180,E1 -20634.291,E2 -20634.291} C_VEL
LIN {X 0,Y 225.056,Z 352.662,A -85,B 0,C 180,E1 -20636.421,E2 -20636.421} C_VEL
LIN {X 0,Y 226.942,Z 347.404,A -85,B 0,C 180,E1 -20637.677,E2 -20637.677} C_VEL
LIN {X 0,Y 228.177,Z 339.553,A -85,B 0,C 180,E1 -20639.523,E2 -20639.523} C_VEL
LIN {X 0,Y 228.873,Z 330.47,A -85,B 0,C 180,E1 -20641.466,E2 -20641.466} C_VEL
LIN {X 0,Y 228.604,Z 319.825,A -85,B 0,C 180,E1 -20643.597,E2 -20643.597} C_VEL
LIN {X 0,Y 226.92,Z 307.074,A -85,B 0,C 180,E1 -20646.045,E2 -20646.045} C_VEL
LIN {X 0,Y 224.501,Z 296.384,A -85,B 0,C 180,E1 -20648.085,E2 -20648.085} C_VEL
LIN {X 0,Y 222.731,Z 290.929,A -85,B 0,C 180,E1 -20649.196,E2 -20649.196} C_VEL
LIN {X 0,Y 221.699,Z 288.52,A -85,B 0,C 180,E1 -20649.752,E2 -20649.752} C_VEL
LIN {X 0,Y 219.976,Z 284.729,A -85,B 0,C 180,E1 -20650.654,E2 -20650.654} C_VEL
LIN {X 0,Y 217.139,Z 280.2,A -85,B 0,C 180,E1 -20651.98,E2 -20651.98} C_VEL
LIN {X 0,Y 216.583,Z 278.245,A -85,B 0,C 180,E1 -20652.374,E2 -20652.374} C_VEL
LIN {X 0,Y 215.974,Z 274.883,A -85,B 0,C 180,E1 -20656.89,E2 -20656.89} C_VEL
LIN {X 0,Y 215.509,Z 271.708,A -85,B 0,C 180,E1 -20661.709,E2 -20661.709} C_VEL
LIN {X 0,Y 215.032,Z 269.201,A -85,B 0,C 180,E1 -20666.244,E2 -20666.244} C_VEL
LIN {X 0,Y 214.726,Z 267.176,A -85,B 0,C 180,E1 -20670.594,E2 -20670.594} C_VEL
LIN {X 0,Y 214.665,Z 266.308,A -85,B 0,C 180,E1 -20672.716,E2 -20672.716} C_VEL
LIN {X 0,Y 214.409,Z 264.955,A -85,B 0,C 180,E1 -20676.835,E2 -20676.835} C_VEL
LIN {X 0,Y 214.245,Z 263.743,A -85,B 0,C 180,E1 -20682.039,E2 -20682.039} C_VEL
LIN {X 0,Y 214.205,Z 263.107,A -85,B 0,C 180,E1 -20686.72,E2 -20686.72} C_VEL
LIN {X 0,Y 214.381,Z 262.853,A -85,B 0,C 180,E1 -20690.563,E2 -20690.563} C_VEL
LIN {X 0,Y 214.427,Z 262.842,A -85,B 0,C 180,E1 -20692.464,E2 -20692.464} C_VEL
LIN {X 0,Y 214.699,Z 263.175,A -85,B 0,C 180,E1 -20698.121,E2 -20698.121} C_VEL
LIN {X 0,Y 214.845,Z 263.404,A -85,B 0,C 180,E1 -20699.997,E2 -20699.997} C_VEL
LIN {X 0,Y 214.577,Z 264.143,A -85,B 0,C 180,E1 -20703.753,E2 -20703.753} C_VEL
LIN {X 0,Y 214.758,Z 265.017,A -85,B 0,C 180,E1 -20707.519,E2 -20707.519} C_VEL
LIN {X 0,Y 214.77,Z 265.852,A -85,B 0,C 180,E1 -20710.167,E2 -20710.167} C_VEL
LIN {X 0,Y 215.993,Z 268.763,A -85,B 0,C 180,E1 -20710.901,E2 -20710.901} C_VEL
LIN {X 0,Y 218.099,Z 271.443,A -85,B 0,C 180,E1 -20711.91,E2 -20711.91} C_VEL
LIN {X 0,Y 220.107,Z 274.951,A -85,B 0,C 180,E1 -20712.963,E2 -20712.963} C_VEL
LIN {X 0,Y 220.803,Z 275.796,A -85,B 0,C 180,E1 -20713.279,E2 -20713.279} C_VEL
LIN {X 0,Y 224.758,Z 283.509,A -85,B 0,C 180,E1 -20715.469,E2 -20715.469} C_VEL
LIN {X 0,Y 228.547,Z 293.024,A -85,B 0,C 180,E1 -20717.906,E2 -20717.906} C_VEL
LIN {X 0,Y 230.956,Z 301.675,A -85,B 0,C 180,E1 -20720.016,E2 -20720.016} C_VEL
LIN {X 0,Y 232.531,Z 310.694,A -85,B 0,C 180,E1 -20722.194,E2 -20722.194} C_VEL
LIN {X 0,Y 232.998,Z 316.619,A -85,B 0,C 180,E1 -20723.668,E2 -20723.668} C_VEL
LIN {X 0,Y 230.68,Z 324.429,A -85,B 0,C 180,E1 -20725.244,E2 -20725.244} C_VEL
LIN {X 0,Y 227.083,Z 334.308,A -85,B 0,C 180,E1 -20727.657,E2 -20727.657} C_VEL
LIN {X 0,Y 223.918,Z 342.3,A -85,B 0,C 180,E1 -20730.141,E2 -20730.141} C_VEL
LIN {X 0,Y 220.944,Z 348.896,A -85,B 0,C 180,E1 -20732.731,E2 -20732.731} C_VEL
LIN {X 0,Y 218.5,Z 354.151,A -85,B 0,C 180,E1 -20735.374,E2 -20735.374} C_VEL
LIN {X 0,Y 216.031,Z 359.077,A -85,B 0,C 180,E1 -20738.671,E2 -20738.671} C_VEL
LIN {X 0,Y 214.638,Z 361.765,A -85,B 0,C 180,E1 -20741.143,E2 -20741.143} C_VEL
LIN {X 0,Y 213.421,Z 363.798,A -85,B 0,C 180,E1 -20743.747,E2 -20743.747} C_VEL
LIN {X 0,Y 212.383,Z 365.149,A -85,B 0,C 180,E1 -20746.714,E2 -20746.714} C_VEL
LIN {X 0,Y 211.768,Z 365.523,A -85,B 0,C 180,E1 -20749.751,E2 -20749.751} C_VEL
LIN {X 0,Y 211.513,Z 364.689,A -85,B 0,C 180,E1 -20753.269,E2 -20753.269} C_VEL
LIN {X 0,Y 211.598,Z 363.038,A -85,B 0,C 180,E1 -20756.128,E2 -20756.128} C_VEL
LIN {X 0,Y 212.154,Z 359.903,A -85,B 0,C 180,E1 -20759.456,E2 -20759.456} C_VEL
LIN {X 0,Y 213.065,Z 355.148,A -85,B 0,C 180,E1 -20762.941,E2 -20762.941} C_VEL
LIN {X 0,Y 214.095,Z 350.133,A -85,B 0,C 180,E1 -20765.698,E2 -20765.698} C_VEL
LIN {X 0,Y 215.518,Z 343.754,A -85,B 0,C 180,E1 -20768.48,E2 -20768.48} C_VEL
LIN {X 0,Y 217.211,Z 336.143,A -85,B 0,C 180,E1 -20771.124,E2 -20771.124} C_VEL
LIN {X 0,Y 219.17,Z 327.192,A -85,B 0,C 180,E1 -20773.624,E2 -20773.624} C_VEL
LIN {X 0,Y 221.179,Z 317.758,A -85,B 0,C 180,E1 -20775.746,E2 -20775.746} C_VEL
LIN {X 0,Y 223.215,Z 306.722,A -85,B 0,C 180,E1 -20777.731,E2 -20777.731} C_VEL
LIN {X 0,Y 223.449,Z 303.831,A -85,B 0,C 180,E1 -20778.204,E2 -20778.204} C_VEL
LIN {X 0,Y 221.643,Z 292.681,A -85,B 0,C 180,E1 -20780.051,E2 -20780.051} C_VEL
LIN {X 0,Y 219.033,Z 281.045,A -85,B 0,C 180,E1 -20781.7,E2 -20781.7} C_VEL
LIN {X 0,Y 215.422,Z 267.945,A -85,B 0,C 180,E1 -20783.269,E2 -20783.269} C_VEL
LIN {X 0,Y 213.468,Z 261.895,A -85,B 0,C 180,E1 -20783.919,E2 -20783.919} C_VEL
LIN {X 0,Y 214.468,Z 261.769,A -85,B 0,C 180,E1 -20790.002,E2 -20790.002} C_VEL
LIN {X 0,Y 214.434,Z 261.775,A -85,B 0,C 180,E1 -20791.88,E2 -20791.88} C_VEL
LIN {X 0,Y 214.216,Z 261.8,A -85,B 0,C 180,E1 -20797.543,E2 -20797.543} C_VEL
LIN {X 0,Y 214.034,Z 261.826,A -85,B 0,C 180,E1 -20801.364,E2 -20801.364} C_VEL
LIN {X 0,Y 213.927,Z 261.835,A -85,B 0,C 180,E1 -20805.239,E2 -20805.239} C_VEL
LIN {X 0,Y 213.872,Z 261.847,A -85,B 0,C 180,E1 -20809.186,E2 -20809.186} C_VEL
LIN {X 0,Y 213.85,Z 261.846,A -85,B 0,C 180,E1 -20813.229,E2 -20813.229} C_VEL
LIN {X 0,Y 213.821,Z 261.852,A -85,B 0,C 180,E1 -20817.453,E2 -20817.453} C_VEL
LIN {X 0,Y 213.772,Z 261.858,A -85,B 0,C 180,E1 -20821.739,E2 -20821.739} C_VEL
LIN {X 0,Y 213.748,Z 261.861,A -85,B 0,C 180,E1 -20826.29,E2 -20826.29} C_VEL
LIN {X 0,Y 213.789,Z 261.854,A -85,B 0,C 180,E1 -20831.11,E2 -20831.11} C_VEL
LIN {X 0,Y 213.805,Z 261.851,A -85,B 0,C 180,E1 -20833.689,E2 -20833.689} C_VEL
LIN {X 0,Y 213.808,Z 261.849,A -85,B 0,C 180,E1 -20836.352,E2 -20836.352} C_VEL
LIN {X 0,Y 213.777,Z 261.851,A -85,B 0,C 180,E1 -20841.349,E2 -20841.349} C_VEL
LIN {X 0,Y 213.768,Z 261.839,A -85,B 0,C 180,E1 -20846.024,E2 -20846.024} C_VEL
LIN {X 0,Y 213.781,Z 261.855,A -85,B 0,C 180,E1 -20850.458,E2 -20850.458} C_VEL
LIN {X 0,Y 213.803,Z 261.849,A -85,B 0,C 180,E1 -20854.706,E2 -20854.706} C_VEL
LIN {X 0,Y 213.815,Z 261.834,A -85,B 0,C 180,E1 -20858.807,E2 -20858.807} C_VEL
LIN {X 0,Y 213.948,Z 261.827,A -85,B 0,C 180,E1 -20862.807,E2 -20862.807} C_VEL
LIN {X 0,Y 213.985,Z 261.828,A -85,B 0,C 180,E1 -20866.712,E2 -20866.712} C_VEL
LIN {X 0,Y 214.145,Z 261.803,A -85,B 0,C 180,E1 -20870.558,E2 -20870.558} C_VEL
LIN {X 0,Y 214.102,Z 261.798,A -85,B 0,C 180,E1 -20874.352,E2 -20874.352} C_VEL
LIN {X 0,Y 214.451,Z 261.77,A -85,B 0,C 180,E1 -20878.125,E2 -20878.125} C_VEL
LIN {X 0,Y 214.554,Z 261.76,A -85,B 0,C 180,E1 -20880.003,E2 -20880.003} C_VEL
LIN {X 0,Y 214.45,Z 261.772,A -85,B 0,C 180,E1 -20881.881,E2 -20881.881} C_VEL
LIN {X 0,Y 214.199,Z 261.79,A -85,B 0,C 180,E1 -20887.544,E2 -20887.544} C_VEL
LIN {X 0,Y 214.007,Z 261.825,A -85,B 0,C 180,E1 -20891.367,E2 -20891.367} C_VEL
LIN {X 0,Y 213.943,Z 261.836,A -85,B 0,C 180,E1 -20895.239,E2 -20895.239} C_VEL
LIN {X 0,Y 213.85,Z 261.837,A -85,B 0,C 180,E1 -20899.189,E2 -20899.189} C_VEL
LIN {X 0,Y 213.858,Z 261.847,A -85,B 0,C 180,E1 -20903.229,E2 -20903.229} C_VEL
LIN {X 0,Y 213.84,Z 261.842,A -85,B 0,C 180,E1 -20907.451,E2 -20907.451} C_VEL
LIN {X 0,Y 213.779,Z 261.855,A -85,B 0,C 180,E1 -20911.739,E2 -20911.739} C_VEL
LIN {X 0,Y 213.755,Z 261.857,A -85,B 0,C 180,E1 -20916.289,E2 -20916.289} C_VEL
LIN {X 0,Y 213.835,Z 261.919,A -85,B 0,C 180,E1 -20917.924,E2 -20917.924} C_VEL
LIN {X 0,Y 214.479,Z 265.6,A -85,B 0,C 180,E1 -20922.203,E2 -20922.203} C_VEL
LIN {X 0,Y 215.219,Z 269.75,A -85,B 0,C 180,E1 -20926.702,E2 -20926.702} C_VEL
LIN {X 0,Y 215.701,Z 272.268,A -85,B 0,C 180,E1 -20929.332,E2 -20929.332} C_VEL
LIN {X 0,Y 215.972,Z 274.726,A -85,B 0,C 180,E1 -20931.807,E2 -20931.807} C_VEL
LIN {X 0,Y 215.64,Z 277.626,A -85,B 0,C 180,E1 -20934.57,E2 -20934.57} C_VEL
LIN {X 0,Y 214.311,Z 282.601,A -85,B 0,C 180,E1 -20939.122,E2 -20939.122} C_VEL
LIN {X 0,Y 216.768,Z 296.298,A -85,B 0,C 180,E1 -20940.323,E2 -20940.323} C_VEL
LIN {X 0,Y 218.43,Z 308.995,A -85,B 0,C 180,E1 -20941.742,E2 -20941.742} C_VEL
LIN {X 0,Y 219.517,Z 320.87,A -85,B 0,C 180,E1 -20943.368,E2 -20943.368} C_VEL
LIN {X 0,Y 219.982,Z 332.271,A -85,B 0,C 180,E1 -20945.245,E2 -20945.245} C_VEL
LIN {X 0,Y 219.95,Z 339.014,A -85,B 0,C 180,E1 -20946.543,E2 -20946.543} C_VEL
LIN {X 0,Y 219.311,Z 342.138,A -85,B 0,C 180,E1 -20947.155,E2 -20947.155} C_VEL
LIN {X 0,Y 218.046,Z 345.12,A -85,B 0,C 180,E1 -20947.746,E2 -20947.746} C_VEL
LIN {X 0,Y 214.471,Z 350.676,A -85,B 0,C 180,E1 -20948.925,E2 -20948.925} C_VEL
LIN {X 0,Y 209.969,Z 357.192,A -85,B 0,C 180,E1 -20950.576,E2 -20950.576} C_VEL
LIN {X 0,Y 208.439,Z 360.939,A -85,B 0,C 180,E1 -20951.745,E2 -20951.745} C_VEL
LIN {X 0,Y 206.762,Z 368.79,A -85,B 0,C 180,E1 -20954.724,E2 -20954.724} C_VEL
LIN {X 0,Y 205.381,Z 375.809,A -85,B 0,C 180,E1 -20958.15,E2 -20958.15} C_VEL
LIN {X 0,Y 204.841,Z 380.453,A -85,B 0,C 180,E1 -20961.116,E2 -20961.116} C_VEL
LIN {X 0,Y 204.721,Z 384.467,A -85,B 0,C 180,E1 -20964.622,E2 -20964.622} C_VEL
LIN {X 0,Y 204.723,Z 386.991,A -85,B 0,C 180,E1 -20968.031,E2 -20968.031} C_VEL
LIN {X 0,Y 204.758,Z 387.87,A -85,B 0,C 180,E1 -20969.998,E2 -20969.998} C_VEL
LIN {X 0,Y 204.672,Z 388.337,A -85,B 0,C 180,E1 -20971.966,E2 -20971.966} C_VEL
LIN {X 0,Y 204.497,Z 387.987,A -85,B 0,C 180,E1 -20975.916,E2 -20975.916} C_VEL
LIN {X 0,Y 204.909,Z 386.094,A -85,B 0,C 180,E1 -20979.872,E2 -20979.872} C_VEL
LIN {X 0,Y 205.42,Z 384.549,A -85,B 0,C 180,E1 -20981.844,E2 -20981.844} C_VEL
LIN {X 0,Y 206.61,Z 381.449,A -85,B 0,C 180,E1 -20984.779,E2 -20984.779} C_VEL
LIN {X 0,Y 208.475,Z 377.342,A -85,B 0,C 180,E1 -20987.66,E2 -20987.66} C_VEL
LIN {X 0,Y 211.252,Z 371.132,A -85,B 0,C 180,E1 -20990.953,E2 -20990.953} C_VEL
LIN {X 0,Y 213.962,Z 364.447,A -85,B 0,C 180,E1 -20993.725,E2 -20993.725} C_VEL
LIN {X 0,Y 217.477,Z 356.266,A -85,B 0,C 180,E1 -20996.379,E2 -20996.379} C_VEL
LIN {X 0,Y 220.659,Z 348.012,A -85,B 0,C 180,E1 -20998.536,E2 -20998.536} C_VEL
LIN {X 0,Y 222.281,Z 338.373,A -85,B 0,C 180,E1 -21000.896,E2 -21000.896} C_VEL
LIN {X 0,Y 222.849,Z 328.281,A -85,B 0,C 180,E1 -21003.137,E2 -21003.137} C_VEL
LIN {X 0,Y 222.481,Z 318.433,A -85,B 0,C 180,E1 -21005.219,E2 -21005.219} C_VEL
LIN {X 0,Y 220.953,Z 306.676,A -85,B 0,C 180,E1 -21007.609,E2 -21007.609} C_VEL
LIN {X 0,Y 218.405,Z 296.049,A -85,B 0,C 180,E1 -21009.86,E2 -21009.86} C_VEL
LIN {X 0,Y 215.365,Z 288.958,A -85,B 0,C 180,E1 -21011.684,E2 -21011.684} C_VEL
LIN {X 0,Y 213.265,Z 285.211,A -85,B 0,C 180,E1 -21012.833,E2 -21012.833} C_VEL
LIN {X 0,Y 212.468,Z 283.455,A -85,B 0,C 180,E1 -21013.301,E2 -21013.301} C_VEL
LIN {X 0,Y 210.298,Z 280.476,A -85,B 0,C 180,E1 -21014.431,E2 -21014.431} C_VEL
LIN {X 0,Y 209.247,Z 277.536,A -85,B 0,C 180,E1 -21015.14,E2 -21015.14} C_VEL
LIN {X 0,Y 208.934,Z 275.722,A -85,B 0,C 180,E1 -21017.73,E2 -21017.73} C_VEL
LIN {X 0,Y 208.435,Z 272.72,A -85,B 0,C 180,E1 -21022.629,E2 -21022.629} C_VEL
LIN {X 0,Y 208.25,Z 271.436,A -85,B 0,C 180,E1 -21024.987,E2 -21024.987} C_VEL
LIN {X 0,Y 207.884,Z 269.279,A -85,B 0,C 180,E1 -21029.526,E2 -21029.526} C_VEL
LIN {X 0,Y 207.654,Z 267.582,A -85,B 0,C 180,E1 -21033.894,E2 -21033.894} C_VEL
LIN {X 0,Y 207.447,Z 266.324,A -85,B 0,C 180,E1 -21038.117,E2 -21038.117} C_VEL
LIN {X 0,Y 207.358,Z 265.418,A -85,B 0,C 180,E1 -21042.237,E2 -21042.237} C_VEL
LIN {X 0,Y 207.306,Z 264.85,A -85,B 0,C 180,E1 -21046.269,E2 -21046.269} C_VEL
LIN {X 0,Y 207.454,Z 264.55,A -85,B 0,C 180,E1 -21050.245,E2 -21050.245} C_VEL
LIN {X 0,Y 207.536,Z 264.521,A -85,B 0,C 180,E1 -21052.212,E2 -21052.212} C_VEL
LIN {X 0,Y 207.769,Z 264.809,A -85,B 0,C 180,E1 -21058.059,E2 -21058.059} C_VEL
LIN {X 0,Y 207.928,Z 265.002,A -85,B 0,C 180,E1 -21059.997,E2 -21059.997} C_VEL
LIN {X 0,Y 207.662,Z 265.742,A -85,B 0,C 180,E1 -21063.878,E2 -21063.878} C_VEL
LIN {X 0,Y 207.82,Z 266.523,A -85,B 0,C 180,E1 -21067.405,E2 -21067.405} C_VEL
LIN {X 0,Y 209.039,Z 269.479,A -85,B 0,C 180,E1 -21068.273,E2 -21068.273} C_VEL
LIN {X 0,Y 211.483,Z 272.248,A -85,B 0,C 180,E1 -21069.561,E2 -21069.561} C_VEL
LIN {X 0,Y 213.523,Z 275.845,A -85,B 0,C 180,E1 -21070.792,E2 -21070.792} C_VEL
LIN {X 0,Y 214.486,Z 277.366,A -85,B 0,C 180,E1 -21071.335,E2 -21071.335} C_VEL
LIN {X 0,Y 218.657,Z 284.971,A -85,B 0,C 180,E1 -21073.825,E2 -21073.825} C_VEL
LIN {X 0,Y 222.491,Z 294.343,A -85,B 0,C 180,E1 -21076.513,E2 -21076.513} C_VEL
LIN {X 0,Y 224.822,Z 302.604,A -85,B 0,C 180,E1 -21078.685,E2 -21078.685} C_VEL
LIN {X 0,Y 226.444,Z 312.239,A -85,B 0,C 180,E1 -21081.195,E2 -21081.195} C_VEL
LIN {X 0,Y 226.845,Z 319.256,A -85,B 0,C 180,E1 -21083.022,E2 -21083.022} C_VEL
LIN {X 0,Y 223.447,Z 328.875,A -85,B 0,C 180,E1 -21085.102,E2 -21085.102} C_VEL
LIN {X 0,Y 219.982,Z 337.532,A -85,B 0,C 180,E1 -21087.464,E2 -21087.464} C_VEL
LIN {X 0,Y 216.899,Z 344.653,A -85,B 0,C 180,E1 -21089.913,E2 -21089.913} C_VEL
LIN {X 0,Y 213.502,Z 351.591,A -85,B 0,C 180,E1 -21092.927,E2 -21092.927} C_VEL
LIN {X 0,Y 211.233,Z 356.05,A -85,B 0,C 180,E1 -21095.451,E2 -21095.451} C_VEL
LIN {X 0,Y 209.269,Z 359.708,A -85,B 0,C 180,E1 -21098.118,E2 -21098.118} C_VEL
LIN {X 0,Y 207.208,Z 363.239,A -85,B 0,C 180,E1 -21101.742,E2 -21101.742} C_VEL
LIN {X 0,Y 206.086,Z 364.793,A -85,B 0,C 180,E1 -21104.266,E2 -21104.266} C_VEL
LIN {X 0,Y 205.261,Z 365.679,A -85,B 0,C 180,E1 -21106.784,E2 -21106.784} C_VEL
LIN {X 0,Y 204.763,Z 365.937,A -85,B 0,C 180,E1 -21109.3,E2 -21109.3} C_VEL
LIN {X 0,Y 204.441,Z 365.399,A -85,B 0,C 180,E1 -21112.242,E2 -21112.242} C_VEL
LIN {X 0,Y 204.468,Z 363.749,A -85,B 0,C 180,E1 -21115.575,E2 -21115.575} C_VEL
LIN {X 0,Y 204.96,Z 360.758,A -85,B 0,C 180,E1 -21119.049,E2 -21119.049} C_VEL
LIN {X 0,Y 205.851,Z 356.267,A -85,B 0,C 180,E1 -21122.574,E2 -21122.574} C_VEL
LIN {X 0,Y 207.072,Z 350.413,A -85,B 0,C 180,E1 -21125.968,E2 -21125.968} C_VEL
LIN {X 0,Y 208.781,Z 343.001,A -85,B 0,C 180,E1 -21129.222,E2 -21129.222} C_VEL
LIN {X 0,Y 210.655,Z 334.891,A -85,B 0,C 180,E1 -21132.027,E2 -21132.027} C_VEL
LIN {X 0,Y 212.879,Z 325.179,A -85,B 0,C 180,E1 -21134.688,E2 -21134.688} C_VEL
LIN {X 0,Y 215.146,Z 314.331,A -85,B 0,C 180,E1 -21137.029,E2 -21137.029} C_VEL
LIN {X 0,Y 216.618,Z 306.43,A -85,B 0,C 180,E1 -21138.421,E2 -21138.421} C_VEL
LIN {X 0,Y 216.006,Z 300.268,A -85,B 0,C 180,E1 -21139.528,E2 -21139.528} C_VEL
LIN {X 0,Y 213.747,Z 288.194,A -85,B 0,C 180,E1 -21141.494,E2 -21141.494} C_VEL
LIN {X 0,Y 210.449,Z 275.086,A -85,B 0,C 180,E1 -21143.29,E2 -21143.29} C_VEL
LIN {X 0,Y 207.352,Z 265.36,A -85,B 0,C 180,E1 -21144.44,E2 -21144.44} C_VEL
LIN {X 0,Y 206.512,Z 262.762,A -85,B 0,C 180,E1 -21144.754,E2 -21144.754} C_VEL
LIN {X 0,Y 207.424,Z 262.646,A -85,B 0,C 180,E1 -21150.002,E2 -21150.002} C_VEL
LIN {X 0,Y 207.371,Z 262.654,A -85,B 0,C 180,E1 -21151.944,E2 -21151.944} C_VEL
LIN {X 0,Y 207.157,Z 262.678,A -85,B 0,C 180,E1 -21157.801,E2 -21157.801} C_VEL
LIN {X 0,Y 206.971,Z 262.704,A -85,B 0,C 180,E1 -21161.758,E2 -21161.758} C_VEL
LIN {X 0,Y 206.867,Z 262.717,A -85,B 0,C 180,E1 -21165.773,E2 -21165.773} C_VEL
LIN {X 0,Y 206.81,Z 262.724,A -85,B 0,C 180,E1 -21169.868,E2 -21169.868} C_VEL
LIN {X 0,Y 206.761,Z 262.73,A -85,B 0,C 180,E1 -21174.074,E2 -21174.074} C_VEL
LIN {X 0,Y 206.736,Z 262.735,A -85,B 0,C 180,E1 -21178.422,E2 -21178.422} C_VEL
LIN {X 0,Y 206.702,Z 262.737,A -85,B 0,C 180,E1 -21182.959,E2 -21182.959} C_VEL
LIN {X 0,Y 206.72,Z 262.734,A -85,B 0,C 180,E1 -21187.734,E2 -21187.734} C_VEL
LIN {X 0,Y 206.719,Z 262.734,A -85,B 0,C 180,E1 -21191.592,E2 -21191.592} C_VEL
LIN {X 0,Y 206.714,Z 262.73,A -85,B 0,C 180,E1 -21195.562,E2 -21195.562} C_VEL
LIN {X 0,Y 206.718,Z 262.734,A -85,B 0,C 180,E1 -21199.767,E2 -21199.767} C_VEL
LIN {X 0,Y 206.723,Z 262.729,A -85,B 0,C 180,E1 -21202.274,E2 -21202.274} C_VEL
LIN {X 0,Y 206.709,Z 262.724,A -85,B 0,C 180,E1 -21207.048,E2 -21207.048} C_VEL
LIN {X 0,Y 206.768,Z 262.729,A -85,B 0,C 180,E1 -21212.1,E2 -21212.1} C_VEL
LIN {X 0,Y 206.788,Z 262.718,A -85,B 0,C 180,E1 -21216.588,E2 -21216.588} C_VEL
LIN {X 0,Y 206.877,Z 262.704,A -85,B 0,C 180,E1 -21222.2,E2 -21222.2} C_VEL
LIN {X 0,Y 206.918,Z 262.71,A -85,B 0,C 180,E1 -21226.249,E2 -21226.249} C_VEL
LIN {X 0,Y 207.105,Z 262.681,A -85,B 0,C 180,E1 -21230.234,E2 -21230.234} C_VEL
LIN {X 0,Y 207.063,Z 262.674,A -85,B 0,C 180,E1 -21234.159,E2 -21234.159} C_VEL
LIN {X 0,Y 207.388,Z 262.648,A -85,B 0,C 180,E1 -21238.061,E2 -21238.061} C_VEL
LIN {X 0,Y 207.519,Z 262.636,A -85,B 0,C 180,E1 -21240.003,E2 -21240.003} C_VEL
LIN {X 0,Y 207.387,Z 262.652,A -85,B 0,C 180,E1 -21241.945,E2 -21241.945} C_VEL
LIN {X 0,Y 207.142,Z 262.668,A -85,B 0,C 180,E1 -21247.803,E2 -21247.803} C_VEL
LIN {X 0,Y 206.933,Z 262.709,A -85,B 0,C 180,E1 -21251.761,E2 -21251.761} C_VEL
LIN {X 0,Y 206.876,Z 262.713,A -85,B 0,C 180,E1 -21255.773,E2 -21255.773} C_VEL
LIN {X 0,Y 206.795,Z 262.719,A -85,B 0,C 180,E1 -21259.871,E2 -21259.871} C_VEL
LIN {X 0,Y 206.774,Z 262.728,A -85,B 0,C 180,E1 -21264.074,E2 -21264.074} C_VEL
LIN {X 0,Y 206.748,Z 262.725,A -85,B 0,C 180,E1 -21268.421,E2 -21268.421} C_VEL
LIN {X 0,Y 206.71,Z 262.737,A -85,B 0,C 180,E1 -21272.959,E2 -21272.959} C_VEL
LIN {X 0,Y 206.805,Z 262.933,A -85,B 0,C 180,E1 -21277.716,E2 -21277.716} C_VEL
LIN {X 0,Y 207.403,Z 266.333,A -85,B 0,C 180,E1 -21281.797,E2 -21281.797} C_VEL
LIN {X 0,Y 208.134,Z 270.387,A -85,B 0,C 180,E1 -21286.38,E2 -21286.38} C_VEL
LIN {X 0,Y 208.822,Z 274.456,A -85,B 0,C 180,E1 -21290.725,E2 -21290.725} C_VEL
LIN {X 0,Y 208.755,Z 277.619,A -85,B 0,C 180,E1 -21293.904,E2 -21293.904} C_VEL
LIN {X 0,Y 207.43,Z 282.193,A -85,B 0,C 180,E1 -21298.251,E2 -21298.251} C_VEL
LIN {X 0,Y 210.027,Z 296.697,A -85,B 0,C 180,E1 -21299.615,E2 -21299.615} C_VEL
LIN {X 0,Y 211.686,Z 309.637,A -85,B 0,C 180,E1 -21301.144,E2 -21301.144} C_VEL
LIN {X 0,Y 212.738,Z 322.311,A -85,B 0,C 180,E1 -21302.984,E2 -21302.984} C_VEL
LIN {X 0,Y 213.118,Z 334.397,A -85,B 0,C 180,E1 -21305.134,E2 -21305.134} C_VEL
LIN {X 0,Y 212.871,Z 340.63,A -85,B 0,C 180,E1 -21306.4,E2 -21306.4} C_VEL
LIN {X 0,Y 210.836,Z 349.794,A -85,B 0,C 180,E1 -21308.487,E2 -21308.487} C_VEL
LIN {X 0,Y 208.912,Z 358.185,A -85,B 0,C 180,E1 -21310.851,E2 -21310.851} C_VEL
LIN {X 0,Y 208.439,Z 360.939,A -85,B 0,C 180,E1 -21311.745,E2 -21311.745} C_VEL
LIN {X 0,Y 207.035,Z 364.551,A -85,B 0,C 180,E1 -21312.975,E2 -21312.975} C_VEL
LIN {X 0,Y 203.027,Z 369.784,A -85,B 0,C 180,E1 -21315.048,E2 -21315.048} C_VEL
LIN {X 0,Y 199.201,Z 374.315,A -85,B 0,C 180,E1 -21317.326,E2 -21317.326} C_VEL
LIN {X 0,Y 198.114,Z 376.831,A -85,B 0,C 180,E1 -21318.842,E2 -21318.842} C_VEL
LIN {X 0,Y 197.672,Z 381.022,A -85,B 0,C 180,E1 -21321.822,E2 -21321.822} C_VEL
LIN {X 0,Y 197.631,Z 384.104,A -85,B 0,C 180,E1 -21324.719,E2 -21324.719} C_VEL
LIN {X 0,Y 197.657,Z 386.458,A -85,B 0,C 180,E1 -21327.96,E2 -21327.96} C_VEL
LIN {X 0,Y 197.69,Z 387.375,A -85,B 0,C 180,E1 -21329.998,E2 -21329.998} C_VEL
LIN {X 0,Y 197.598,Z 387.878,A -85,B 0,C 180,E1 -21332.036,E2 -21332.036} C_VEL
LIN {X 0,Y 197.412,Z 387.915,A -85,B 0,C 180,E1 -21334.541,E2 -21334.541} C_VEL
LIN {X 0,Y 197.565,Z 386.926,A -85,B 0,C 180,E1 -21338.178,E2 -21338.178} C_VEL
LIN {X 0,Y 198.447,Z 384.352,A -85,B 0,C 180,E1 -21342.266,E2 -21342.266} C_VEL
LIN {X 0,Y 199.727,Z 381.319,A -85,B 0,C 180,E1 -21345.3,E2 -21345.3} C_VEL
LIN {X 0,Y 201.676,Z 377.299,A -85,B 0,C 180,E1 -21348.276,E2 -21348.276} C_VEL
LIN {X 0,Y 204.181,Z 372.214,A -85,B 0,C 180,E1 -21351.185,E2 -21351.185} C_VEL
LIN {X 0,Y 206.968,Z 365.927,A -85,B 0,C 180,E1 -21354.045,E2 -21354.045} C_VEL
LIN {X 0,Y 210.528,Z 358.174,A -85,B 0,C 180,E1 -21356.784,E2 -21356.784} C_VEL
LIN {X 0,Y 213.901,Z 350.353,A -85,B 0,C 180,E1 -21358.986,E2 -21358.986} C_VEL
LIN {X 0,Y 215.198,Z 345.008,A -85,B 0,C 180,E1 -21360.409,E2 -21360.409} C_VEL
LIN {X 0,Y 216.517,Z 336.146,A -85,B 0,C 180,E1 -21362.61,E2 -21362.61} C_VEL
LIN {X 0,Y 216.945,Z 326.407,A -85,B 0,C 180,E1 -21364.876,E2 -21364.876} C_VEL
LIN {X 0,Y 216.321,Z 315.403,A -85,B 0,C 180,E1 -21367.316,E2 -21367.316} C_VEL
LIN {X 0,Y 214.779,Z 304.905,A -85,B 0,C 180,E1 -21369.637,E2 -21369.637} C_VEL
LIN {X 0,Y 213.565,Z 299.896,A -85,B 0,C 180,E1 -21370.806,E2 -21370.806} C_VEL
LIN {X 0,Y 211.453,Z 294.435,A -85,B 0,C 180,E1 -21372.306,E2 -21372.306} C_VEL
LIN {X 0,Y 209.109,Z 289.698,A -85,B 0,C 180,E1 -21373.819,E2 -21373.819} C_VEL
LIN {X 0,Y 206.27,Z 284.798,A -85,B 0,C 180,E1 -21375.57,E2 -21375.57} C_VEL
LIN {X 0,Y 205.529,Z 283.095,A -85,B 0,C 180,E1 -21376.08,E2 -21376.08} C_VEL
LIN {X 0,Y 203.055,Z 279.844,A -85,B 0,C 180,E1 -21377.597,E2 -21377.597} C_VEL
LIN {X 0,Y 201.864,Z 276.646,A -85,B 0,C 180,E1 -21378.583,E2 -21378.583} C_VEL
LIN {X 0,Y 201.453,Z 273.728,A -85,B 0,C 180,E1 -21383.622,E2 -21383.622} C_VEL
LIN {X 0,Y 201.019,Z 271.44,A -85,B 0,C 180,E1 -21388.367,E2 -21388.367} C_VEL
LIN {X 0,Y 200.789,Z 269.606,A -85,B 0,C 180,E1 -21392.93,E2 -21392.93} C_VEL
LIN {X 0,Y 200.563,Z 268.247,A -85,B 0,C 180,E1 -21397.325,E2 -21397.325} C_VEL
LIN {X 0,Y 200.47,Z 267.256,A -85,B 0,C 180,E1 -21401.605,E2 -21401.605} C_VEL
LIN {X 0,Y 200.4,Z 266.63,A -85,B 0,C 180,E1 -21405.786,E2 -21405.786} C_VEL
LIN {X 0,Y 200.535,Z 266.277,A -85,B 0,C 180,E1 -21409.905,E2 -21409.905} C_VEL
LIN {X 0,Y 200.632,Z 266.204,A -85,B 0,C 180,E1 -21411.942,E2 -21411.942} C_VEL
LIN {X 0,Y 200.853,Z 266.436,A -85,B 0,C 180,E1 -21417.992,E2 -21417.992} C_VEL
LIN {X 0,Y 201.038,Z 266.628,A -85,B 0,C 180,E1 -21419.997,E2 -21419.997} C_VEL
LIN {X 0,Y 200.771,Z 267.49,A -85,B 0,C 180,E1 -21424.074,E2 -21424.074} C_VEL
LIN {X 0,Y 201.957,Z 270.238,A -85,B 0,C 180,E1 -21425.05,E2 -21425.05} C_VEL
LIN {X 0,Y 204.791,Z 273.044,A -85,B 0,C 180,E1 -21426.79,E2 -21426.79} C_VEL
LIN {X 0,Y 206.461,Z 276.2,A -85,B 0,C 180,E1 -21428.007,E2 -21428.007} C_VEL
LIN {X 0,Y 207.752,Z 277.575,A -85,B 0,C 180,E1 -21428.753,E2 -21428.753} C_VEL
LIN {X 0,Y 209.752,Z 281.349,A -85,B 0,C 180,E1 -21430.128,E2 -21430.128} C_VEL
LIN {X 0,Y 213.519,Z 288.576,A -85,B 0,C 180,E1 -21432.708,E2 -21432.708} C_VEL
LIN {X 0,Y 216.553,Z 295.951,A -85,B 0,C 180,E1 -21435.045,E2 -21435.045} C_VEL
LIN {X 0,Y 219.026,Z 304.865,A -85,B 0,C 180,E1 -21437.624,E2 -21437.624} C_VEL
LIN {X 0,Y 220.477,Z 313.95,A -85,B 0,C 180,E1 -21440.158,E2 -21440.158} C_VEL
LIN {X 0,Y 220.829,Z 320.376,A -85,B 0,C 180,E1 -21441.963,E2 -21441.963} C_VEL
LIN {X 0,Y 219.307,Z 325.152,A -85,B 0,C 180,E1 -21443.024,E2 -21443.024} C_VEL
LIN {X 0,Y 215.5,Z 334.72,A -85,B 0,C 180,E1 -21445.442,E2 -21445.442} C_VEL
LIN {X 0,Y 212.225,Z 342.043,A -85,B 0,C 180,E1 -21447.764,E2 -21447.764} C_VEL
LIN {X 0,Y 209.131,Z 348.372,A -85,B 0,C 180,E1 -21450.267,E2 -21450.267} C_VEL
LIN {X 0,Y 206.124,Z 353.966,A -85,B 0,C 180,E1 -21453.057,E2 -21453.057} C_VEL
LIN {X 0,Y 203.674,Z 358.353,A -85,B 0,C 180,E1 -21455.912,E2 -21455.912} C_VEL
LIN {X 0,Y 201.13,Z 362.582,A -85,B 0,C 180,E1 -21459.763,E2 -21459.763} C_VEL
LIN {X 0,Y 199.776,Z 364.523,A -85,B 0,C 180,E1 -21462.377,E2 -21462.377} C_VEL
LIN {X 0,Y 198.719,Z 365.737,A -85,B 0,C 180,E1 -21465.013,E2 -21465.013} C_VEL
LIN {X 0,Y 197.842,Z 366.333,A -85,B 0,C 180,E1 -21468.239,E2 -21468.239} C_VEL
LIN {X 0,Y 197.402,Z 365.922,A -85,B 0,C 180,E1 -21471.554,E2 -21471.554} C_VEL
LIN {X 0,Y 197.348,Z 364.242,A -85,B 0,C 180,E1 -21475.267,E2 -21475.267} C_VEL
LIN {X 0,Y 197.751,Z 361.644,A -85,B 0,C 180,E1 -21478.527,E2 -21478.527} C_VEL
LIN {X 0,Y 198.393,Z 358.537,A -85,B 0,C 180,E1 -21481.294,E2 -21481.294} C_VEL
LIN {X 0,Y 199.546,Z 352.988,A -85,B 0,C 180,E1 -21485.001,E2 -21485.001} C_VEL
LIN {X 0,Y 201.168,Z 345.968,A -85,B 0,C 180,E1 -21488.482,E2 -21488.482} C_VEL
LIN {X 0,Y 202.917,Z 338.703,A -85,B 0,C 180,E1 -21491.317,E2 -21491.317} C_VEL
LIN {X 0,Y 205.044,Z 329.797,A -85,B 0,C 180,E1 -21494.088,E2 -21494.088} C_VEL
LIN {X 0,Y 207.431,Z 319.28,A -85,B 0,C 180,E1 -21496.667,E2 -21496.667} C_VEL
LIN {X 0,Y 209.531,Z 308.998,A -85,B 0,C 180,E1 -21498.677,E2 -21498.677} C_VEL
LIN {X 0,Y 209.814,Z 305.692,A -85,B 0,C 180,E1 -21499.262,E2 -21499.262} C_VEL
LIN {X 0,Y 208.065,Z 294.669,A -85,B 0,C 180,E1 -21501.269,E2 -21501.269} C_VEL
LIN {X 0,Y 205.513,Z 283.062,A -85,B 0,C 180,E1 -21503.079,E2 -21503.079} C_VEL
LIN {X 0,Y 202.166,Z 270.85,A -85,B 0,C 180,E1 -21504.704,E2 -21504.704} C_VEL
LIN {X 0,Y 199.534,Z 263.63,A -85,B 0,C 180,E1 -21505.646,E2 -21505.646} C_VEL
LIN {X 0,Y 200.379,Z 263.524,A -85,B 0,C 180,E1 -21510.002,E2 -21510.002} C_VEL
LIN {X 0,Y 200.31,Z 263.534,A -85,B 0,C 180,E1 -21512.013,E2 -21512.013} C_VEL
LIN {X 0,Y 200.1,Z 263.557,A -85,B 0,C 180,E1 -21518.078,E2 -21518.078} C_VEL
LIN {X 0,Y 199.903,Z 263.584,A -85,B 0,C 180,E1 -21522.18,E2 -21522.18} C_VEL
LIN {X 0,Y 199.805,Z 263.596,A -85,B 0,C 180,E1 -21526.346,E2 -21526.346} C_VEL
LIN {X 0,Y 199.739,Z 263.604,A -85,B 0,C 180,E1 -21530.603,E2 -21530.603} C_VEL
LIN {X 0,Y 199.669,Z 263.618,A -85,B 0,C 180,E1 -21534.987,E2 -21534.987} C_VEL
LIN {X 0,Y 199.668,Z 263.615,A -85,B 0,C 180,E1 -21539.526,E2 -21539.526} C_VEL
LIN {X 0,Y 199.658,Z 263.618,A -85,B 0,C 180,E1 -21542.356,E2 -21542.356} C_VEL
LIN {X 0,Y 199.647,Z 263.619,A -85,B 0,C 180,E1 -21546.76,E2 -21546.76} C_VEL
LIN {X 0,Y 199.673,Z 263.609,A -85,B 0,C 180,E1 -21549.315,E2 -21549.315} C_VEL
LIN {X 0,Y 199.658,Z 263.616,A -85,B 0,C 180,E1 -21552.342,E2 -21552.342} C_VEL
LIN {X 0,Y 199.662,Z 263.609,A -85,B 0,C 180,E1 -21555.257,E2 -21555.257} C_VEL
LIN {X 0,Y 199.659,Z 263.614,A -85,B 0,C 180,E1 -21558.03,E2 -21558.03} C_VEL
LIN {X 0,Y 199.677,Z 263.609,A -85,B 0,C 180,E1 -21560.747,E2 -21560.747} C_VEL
LIN {X 0,Y 199.633,Z 263.596,A -85,B 0,C 180,E1 -21565.722,E2 -21565.722} C_VEL
LIN {X 0,Y 199.704,Z 263.598,A -85,B 0,C 180,E1 -21568.142,E2 -21568.142} C_VEL
LIN {X 0,Y 199.688,Z 263.61,A -85,B 0,C 180,E1 -21572.776,E2 -21572.776} C_VEL
LIN {X 0,Y 199.74,Z 263.594,A -85,B 0,C 180,E1 -21577.233,E2 -21577.233} C_VEL
LIN {X 0,Y 199.8,Z 263.582,A -85,B 0,C 180,E1 -21581.761,E2 -21581.761} C_VEL
LIN {X 0,Y 199.853,Z 263.589,A -85,B 0,C 180,E1 -21585.753,E2 -21585.753} C_VEL
LIN {X 0,Y 200.028,Z 263.565,A -85,B 0,C 180,E1 -21589.885,E2 -21589.885} C_VEL
LIN {X 0,Y 200.025,Z 263.549,A -85,B 0,C 180,E1 -21593.953,E2 -21593.953} C_VEL
LIN {X 0,Y 200.327,Z 263.527,A -85,B 0,C 180,E1 -21597.993,E2 -21597.993} C_VEL
LIN {X 0,Y 200.484,Z 263.512,A -85,B 0,C 180,E1 -21600.003,E2 -21600.003} C_VEL
LIN {X 0,Y 200.028,Z 263.564,A -85,B 0,C 180,E1 -21604.033,E2 -21604.033} C_VEL
LIN {X 0,Y 200.092,Z 263.546,A -85,B 0,C 180,E1 -21608.08,E2 -21608.08} C_VEL
LIN {X 0,Y 199.883,Z 263.586,A -85,B 0,C 180,E1 -21612.182,E2 -21612.182} C_VEL
LIN {X 0,Y 199.814,Z 263.591,A -85,B 0,C 180,E1 -21616.346,E2 -21616.346} C_VEL
LIN {X 0,Y 199.711,Z 263.602,A -85,B 0,C 180,E1 -21620.607,E2 -21620.607} C_VEL
LIN {X 0,Y 199.684,Z 263.612,A -85,B 0,C 180,E1 -21624.986,E2 -21624.986} C_VEL
LIN {X 0,Y 199.676,Z 263.611,A -85,B 0,C 180,E1 -21629.525,E2 -21629.525} C_VEL
LIN {X 0,Y 199.682,Z 263.611,A -85,B 0,C 180,E1 -21632.357,E2 -21632.357} C_VEL
LIN {X 0,Y 199.731,Z 263.719,A -85,B 0,C 180,E1 -21637.216,E2 -21637.216} C_VEL
LIN {X 0,Y 200.395,Z 267.391,A -85,B 0,C 180,E1 -21641.789,E2 -21641.789} C_VEL
LIN {X 0,Y 201.23,Z 272.037,A -85,B 0,C 180,E1 -21647.178,E2 -21647.178} C_VEL
LIN {X 0,Y 201.773,Z 275.67,A -85,B 0,C 180,E1 -21651.171,E2 -21651.171} C_VEL
LIN {X 0,Y 201.713,Z 278.098,A -85,B 0,C 180,E1 -21653.677,E2 -21653.677} C_VEL
LIN {X 0,Y 200.598,Z 281.867,A -85,B 0,C 180,E1 -21657.4,E2 -21657.4} C_VEL
LIN {X 0,Y 203.003,Z 295.504,A -85,B 0,C 180,E1 -21658.691,E2 -21658.691} C_VEL
LIN {X 0,Y 204.704,Z 308.099,A -85,B 0,C 180,E1 -21660.215,E2 -21660.215} C_VEL
LIN {X 0,Y 205.704,Z 320.209,A -85,B 0,C 180,E1 -21661.996,E2 -21661.996} C_VEL
LIN {X 0,Y 206.146,Z 331.303,A -85,B 0,C 180,E1 -21663.962,E2 -21663.962} C_VEL
LIN {X 0,Y 206.044,Z 340.281,A -85,B 0,C 180,E1 -21665.836,E2 -21665.836} C_VEL
LIN {X 0,Y 203.701,Z 350.506,A -85,B 0,C 180,E1 -21668.28,E2 -21668.28} C_VEL
LIN {X 0,Y 201.837,Z 358.628,A -85,B 0,C 180,E1 -21670.7,E2 -21670.7} C_VEL
LIN {X 0,Y 200.108,Z 366.671,A -85,B 0,C 180,E1 -21673.68,E2 -21673.68} C_VEL
LIN {X 0,Y 198.71,Z 373.148,A -85,B 0,C 180,E1 -21676.707,E2 -21676.707} C_VEL
LIN {X 0,Y 198.114,Z 376.831,A -85,B 0,C 180,E1 -21678.842,E2 -21678.842} C_VEL
LIN {X 0,Y 197.162,Z 379.152,A -85,B 0,C 180,E1 -21680.401,E2 -21680.401} C_VEL
LIN {X 0,Y 194.033,Z 382.213,A -85,B 0,C 180,E1 -21683.014,E2 -21683.014} C_VEL
LIN {X 0,Y 191.573,Z 384.113,A -85,B 0,C 180,E1 -21685.203,E2 -21685.203} C_VEL
LIN {X 0,Y 190.602,Z 385.318,A -85,B 0,C 180,E1 -21686.927,E2 -21686.927} C_VEL
LIN {X 0,Y 190.559,Z 385.665,A -85,B 0,C 180,E1 -21687.512,E2 -21687.512} C_VEL
LIN {X 0,Y 190.623,Z 386.869,A -85,B 0,C 180,E1 -21689.998,E2 -21689.998} C_VEL
LIN {X 0,Y 190.501,Z 387.41,A -85,B 0,C 180,E1 -21692.112,E2 -21692.112} C_VEL
LIN {X 0,Y 190.337,Z 387.554,A -85,B 0,C 180,E1 -21694.447,E2 -21694.447} C_VEL
LIN {X 0,Y 190.509,Z 386.623,A -85,B 0,C 180,E1 -21698.484,E2 -21698.484} C_VEL
LIN {X 0,Y 191.473,Z 384.132,A -85,B 0,C 180,E1 -21702.72,E2 -21702.72} C_VEL
LIN {X 0,Y 192.867,Z 381.199,A -85,B 0,C 180,E1 -21705.858,E2 -21705.858} C_VEL
LIN {X 0,Y 194.906,Z 377.296,A -85,B 0,C 180,E1 -21708.935,E2 -21708.935} C_VEL
LIN {X 0,Y 197.558,Z 372.324,A -85,B 0,C 180,E1 -21711.931,E2 -21711.931} C_VEL
LIN {X 0,Y 200.496,Z 366.156,A -85,B 0,C 180,E1 -21714.872,E2 -21714.872} C_VEL
LIN {X 0,Y 204.22,Z 358.577,A -85,B 0,C 180,E1 -21717.681,E2 -21717.681} C_VEL
LIN {X 0,Y 207.729,Z 350.944,A -85,B 0,C 180,E1 -21719.933,E2 -21719.933} C_VEL
LIN {X 0,Y 209.81,Z 342.068,A -85,B 0,C 180,E1 -21722.406,E2 -21722.406} C_VEL
LIN {X 0,Y 210.806,Z 333.802,A -85,B 0,C 180,E1 -21724.522,E2 -21724.522} C_VEL
LIN {X 0,Y 211.079,Z 323.762,A -85,B 0,C 180,E1 -21726.953,E2 -21726.953} C_VEL
LIN {X 0,Y 210.443,Z 313.447,A -85,B 0,C 180,E1 -21729.382,E2 -21729.382} C_VEL
LIN {X 0,Y 208.823,Z 304.139,A -85,B 0,C 180,E1 -21731.653,E2 -21731.653} C_VEL
LIN {X 0,Y 207.071,Z 299.245,A -85,B 0,C 180,E1 -21733.133,E2 -21733.133} C_VEL
LIN {X 0,Y 204.976,Z 294.556,A -85,B 0,C 180,E1 -21734.709,E2 -21734.709} C_VEL
LIN {X 0,Y 202.555,Z 289.926,A -85,B 0,C 180,E1 -21736.464,E2 -21736.464} C_VEL
LIN {X 0,Y 201.86,Z 288.572,A -85,B 0,C 180,E1 -21736.979,E2 -21736.979} C_VEL
LIN {X 0,Y 199.671,Z 285.096,A -85,B 0,C 180,E1 -21738.546,E2 -21738.546} C_VEL
LIN {X 0,Y 198.486,Z 282.444,A -85,B 0,C 180,E1 -21739.531,E2 -21739.531} C_VEL
LIN {X 0,Y 195.638,Z 278.729,A -85,B 0,C 180,E1 -21741.704,E2 -21741.704} C_VEL
LIN {X 0,Y 194.555,Z 275.685,A -85,B 0,C 180,E1 -21742.873,E2 -21742.873} C_VEL
LIN {X 0,Y 194.21,Z 273.615,A -85,B 0,C 180,E1 -21747.121,E2 -21747.121} C_VEL
LIN {X 0,Y 193.927,Z 271.648,A -85,B 0,C 180,E1 -21751.889,E2 -21751.889} C_VEL
LIN {X 0,Y 193.696,Z 270.185,A -85,B 0,C 180,E1 -21756.474,E2 -21756.474} C_VEL
LIN {X 0,Y 193.559,Z 269.107,A -85,B 0,C 180,E1 -21760.923,E2 -21760.923} C_VEL
LIN {X 0,Y 193.511,Z 268.422,A -85,B 0,C 180,E1 -21765.269,E2 -21765.269} C_VEL
LIN {X 0,Y 193.621,Z 268.001,A -85,B 0,C 180,E1 -21769.54,E2 -21769.54} C_VEL
LIN {X 0,Y 193.72,Z 267.899,A -85,B 0,C 180,E1 -21771.653,E2 -21771.653} C_VEL
LIN {X 0,Y 193.923,Z 268.066,A -85,B 0,C 180,E1 -21777.92,E2 -21777.92} C_VEL
LIN {X 0,Y 194.123,Z 268.285,A -85,B 0,C 180,E1 -21780.062,E2 -21780.062} C_VEL
LIN {X 0,Y 195.133,Z 270.896,A -85,B 0,C 180,E1 -21781.158,E2 -21781.158} C_VEL
LIN {X 0,Y 197.716,Z 273.593,A -85,B 0,C 180,E1 -21783.18,E2 -21783.18} C_VEL
LIN {X 0,Y 199.715,Z 277.222,A -85,B 0,C 180,E1 -21784.917,E2 -21784.917} C_VEL
LIN {X 0,Y 201.362,Z 278.82,A -85,B 0,C 180,E1 -21786.007,E2 -21786.007} C_VEL
LIN {X 0,Y 203.308,Z 282.323,A -85,B 0,C 180,E1 -21787.556,E2 -21787.556} C_VEL
LIN {X 0,Y 206.297,Z 287.552,A -85,B 0,C 180,E1 -21789.804,E2 -21789.804} C_VEL
LIN {X 0,Y 210.055,Z 295.881,A -85,B 0,C 180,E1 -21792.894,E2 -21792.894} C_VEL
LIN {X 0,Y 212.48,Z 303.428,A -85,B 0,C 180,E1 -21795.34,E2 -21795.34} C_VEL
LIN {X 0,Y 214.187,Z 312.348,A -85,B 0,C 180,E1 -21798.061,E2 -21798.061} C_VEL
LIN {X 0,Y 214.824,Z 320.807,A -85,B 0,C 180,E1 -21800.587,E2 -21800.587} C_VEL
LIN {X 0,Y 214.592,Z 323.583,A -85,B 0,C 180,E1 -21801.386,E2 -21801.386} C_VEL
LIN {X 0,Y 210.499,Z 333.552,A -85,B 0,C 180,E1 -21803.831,E2 -21803.831} C_VEL
LIN {X 0,Y 206.975,Z 341.125,A -85,B 0,C 180,E1 -21806.191,E2 -21806.191} C_VEL
LIN {X 0,Y 203.391,Z 348.116,A -85,B 0,C 180,E1 -21808.927,E2 -21808.927} C_VEL
LIN {X 0,Y 200.117,Z 353.862,A -85,B 0,C 180,E1 -21811.785,E2 -21811.785} C_VEL
LIN {X 0,Y 197.22,Z 358.701,A -85,B 0,C 180,E1 -21814.958,E2 -21814.958} C_VEL
LIN {X 0,Y 194.397,Z 363.045,A -85,B 0,C 180,E1 -21819.038,E2 -21819.038} C_VEL
LIN {X 0,Y 192.352,Z 365.625,A -85,B 0,C 180,E1 -21823.054,E2 -21823.054} C_VEL
LIN {X 0,Y 190.915,Z 366.738,A -85,B 0,C 180,E1 -21827.407,E2 -21827.407} C_VEL
LIN {X 0,Y 190.348,Z 366.362,A -85,B 0,C 180,E1 -21831.124,E2 -21831.124} C_VEL
LIN {X 0,Y 190.205,Z 365.052,A -85,B 0,C 180,E1 -21834.373,E2 -21834.373} C_VEL
LIN {X 0,Y 190.554,Z 362.438,A -85,B 0,C 180,E1 -21838.018,E2 -21838.018} C_VEL
LIN {X 0,Y 191.42,Z 358.396,A -85,B 0,C 180,E1 -21841.774,E2 -21841.774} C_VEL
LIN {X 0,Y 192.381,Z 353.786,A -85,B 0,C 180,E1 -21844.931,E2 -21844.931} C_VEL
LIN {X 0,Y 193.853,Z 347.653,A -85,B 0,C 180,E1 -21848.188,E2 -21848.188} C_VEL
LIN {X 0,Y 195.571,Z 340.652,A -85,B 0,C 180,E1 -21851.132,E2 -21851.132} C_VEL
LIN {X 0,Y 197.842,Z 331.46,A -85,B 0,C 180,E1 -21854.206,E2 -21854.206} C_VEL
LIN {X 0,Y 200.253,Z 321.508,A -85,B 0,C 180,E1 -21856.817,E2 -21856.817} C_VEL
LIN {X 0,Y 202.526,Z 311.034,A -85,B 0,C 180,E1 -21858.999,E2 -21858.999} C_VEL
LIN {X 0,Y 203.072,Z 308.111,A -85,B 0,C 180,E1 -21859.534,E2 -21859.534} C_VEL
LIN {X 0,Y 201.921,Z 299.343,A -85,B 0,C 180,E1 -21861.251,E2 -21861.251} C_VEL
LIN {X 0,Y 199.884,Z 288.901,A -85,B 0,C 180,E1 -21863.062,E2 -21863.062} C_VEL
LIN {X 0,Y 196.783,Z 276.261,A -85,B 0,C 180,E1 -21864.943,E2 -21864.943} C_VEL
LIN {X 0,Y 193.303,Z 266.905,A -85,B 0,C 180,E1 -21866.256,E2 -21866.256} C_VEL
LIN {X 0,Y 192.602,Z 264.494,A -85,B 0,C 180,E1 -21866.603,E2 -21866.603} C_VEL
LIN {X 0,Y 193.331,Z 264.402,A -85,B 0,C 180,E1 -21870.002,E2 -21870.002} C_VEL
LIN {X 0,Y 193.252,Z 264.413,A -85,B 0,C 180,E1 -21872.086,E2 -21872.086} C_VEL
LIN {X 0,Y 193.051,Z 264.435,A -85,B 0,C 180,E1 -21878.375,E2 -21878.375} C_VEL
LIN {X 0,Y 192.843,Z 264.464,A -85,B 0,C 180,E1 -21882.633,E2 -21882.633} C_VEL
LIN {X 0,Y 192.773,Z 264.476,A -85,B 0,C 180,E1 -21888.59,E2 -21888.59} C_VEL
LIN {X 0,Y 192.662,Z 264.487,A -85,B 0,C 180,E1 -21894.232,E2 -21894.232} C_VEL
LIN {X 0,Y 192.643,Z 264.491,A -85,B 0,C 180,E1 -21898.896,E2 -21898.896} C_VEL
LIN {X 0,Y 192.594,Z 264.493,A -85,B 0,C 180,E1 -21903.189,E2 -21903.189} C_VEL
LIN {X 0,Y 192.595,Z 264.495,A -85,B 0,C 180,E1 -21908.344,E2 -21908.344} C_VEL
LIN {X 0,Y 192.601,Z 264.493,A -85,B 0,C 180,E1 -21913.136,E2 -21913.136} C_VEL
LIN {X 0,Y 192.6,Z 264.494,A -85,B 0,C 180,E1 -21916.873,E2 -21916.873} C_VEL
LIN {X 0,Y 192.598,Z 264.489,A -85,B 0,C 180,E1 -21921.664,E2 -21921.664} C_VEL
LIN {X 0,Y 192.6,Z 264.478,A -85,B 0,C 180,E1 -21926.819,E2 -21926.819} C_VEL
LIN {X 0,Y 192.666,Z 264.484,A -85,B 0,C 180,E1 -21931.696,E2 -21931.696} C_VEL
LIN {X 0,Y 192.708,Z 264.472,A -85,B 0,C 180,E1 -21936.353,E2 -21936.353} C_VEL
LIN {X 0,Y 192.736,Z 264.46,A -85,B 0,C 180,E1 -21941.462,E2 -21941.462} C_VEL
LIN {X 0,Y 192.777,Z 264.468,A -85,B 0,C 180,E1 -21945.218,E2 -21945.218} C_VEL
LIN {X 0,Y 192.951,Z 264.448,A -85,B 0,C 180,E1 -21949.57,E2 -21949.57} C_VEL
LIN {X 0,Y 192.988,Z 264.426,A -85,B 0,C 180,E1 -21953.731,E2 -21953.731} C_VEL
LIN {X 0,Y 193.269,Z 264.405,A -85,B 0,C 180,E1 -21957.919,E2 -21957.919} C_VEL
LIN {X 0,Y 193.448,Z 264.389,A -85,B 0,C 180,E1 -21960.003,E2 -21960.003} C_VEL
LIN {X 0,Y 192.973,Z 264.442,A -85,B 0,C 180,E1 -21964.18,E2 -21964.18} C_VEL
LIN {X 0,Y 193.041,Z 264.425,A -85,B 0,C 180,E1 -21968.377,E2 -21968.377} C_VEL
LIN {X 0,Y 192.811,Z 264.466,A -85,B 0,C 180,E1 -21972.636,E2 -21972.636} C_VEL
LIN {X 0,Y 192.768,Z 264.468,A -85,B 0,C 180,E1 -21976.961,E2 -21976.961} C_VEL
LIN {X 0,Y 192.648,Z 264.485,A -85,B 0,C 180,E1 -21981.399,E2 -21981.399} C_VEL
LIN {X 0,Y 192.675,Z 264.484,A -85,B 0,C 180,E1 -21984.226,E2 -21984.226} C_VEL
LIN {X 0,Y 192.655,Z 264.481,A -85,B 0,C 180,E1 -21988.89,E2 -21988.89} C_VEL
LIN {X 0,Y 192.608,Z 264.494,A -85,B 0,C 180,E1 -21993.187,E2 -21993.187} C_VEL
LIN {X 0,Y 192.707,Z 264.643,A -85,B 0,C 180,E1 -21996.896,E2 -21996.896} C_VEL
LIN {X 0,Y 193.433,Z 268.74,A -85,B 0,C 180,E1 -22002.151,E2 -22002.151} C_VEL
LIN {X 0,Y 194.073,Z 272.357,A -85,B 0,C 180,E1 -22006.521,E2 -22006.521} C_VEL
LIN {X 0,Y 194.69,Z 276.113,A -85,B 0,C 180,E1 -22010.82,E2 -22010.82} C_VEL
LIN {X 0,Y 194.748,Z 277.716,A -85,B 0,C 180,E1 -22012.559,E2 -22012.559} C_VEL
LIN {X 0,Y 193.759,Z 281.466,A -85,B 0,C 180,E1 -22016.449,E2 -22016.449} C_VEL
LIN {X 0,Y 196.15,Z 295.133,A -85,B 0,C 180,E1 -22017.812,E2 -22017.812} C_VEL
LIN {X 0,Y 197.742,Z 306.594,A -85,B 0,C 180,E1 -22019.251,E2 -22019.251} C_VEL
LIN {X 0,Y 198.805,Z 319.314,A -85,B 0,C 180,E1 -22021.17,E2 -22021.17} C_VEL
LIN {X 0,Y 199.272,Z 330.859,A -85,B 0,C 180,E1 -22023.275,E2 -22023.275} C_VEL
LIN {X 0,Y 199.192,Z 339.897,A -85,B 0,C 180,E1 -22025.228,E2 -22025.228} C_VEL
LIN {X 0,Y 197.146,Z 349.071,A -85,B 0,C 180,E1 -22027.465,E2 -22027.465} C_VEL
LIN {X 0,Y 194.971,Z 357.838,A -85,B 0,C 180,E1 -22030.119,E2 -22030.119} C_VEL
LIN {X 0,Y 193.248,Z 365.663,A -85,B 0,C 180,E1 -22033.084,E2 -22033.084} C_VEL
LIN {X 0,Y 191.752,Z 372.251,A -85,B 0,C 180,E1 -22036.216,E2 -22036.216} C_VEL
LIN {X 0,Y 190.923,Z 377.501,A -85,B 0,C 180,E1 -22039.392,E2 -22039.392} C_VEL
LIN {X 0,Y 190.522,Z 381.546,A -85,B 0,C 180,E1 -22042.58,E2 -22042.58} C_VEL
LIN {X 0,Y 190.521,Z 384.506,A -85,B 0,C 180,E1 -22045.767,E2 -22045.767} C_VEL
LIN {X 0,Y 190.559,Z 385.665,A -85,B 0,C 180,E1 -22047.512,E2 -22047.512} C_VEL
LIN {X 0,Y 189.939,Z 386.616,A -85,B 0,C 180,E1 -22049.252,E2 -22049.252} C_VEL
LIN {X 0,Y 188.304,Z 387.18,A -85,B 0,C 180,E1 -22050.975,E2 -22050.975} C_VEL
LIN {X 0,Y 184.411,Z 387.322,A -85,B 0,C 180,E1 -22054.487,E2 -22054.487} C_VEL
LIN {X 0,Y 183.355,Z 386.992,A -85,B 0,C 180,E1 -22056.332,E2 -22056.332} C_VEL
LIN {X 0,Y 183.293,Z 386.832,A -85,B 0,C 180,E1 -22056.957,E2 -22056.957} C_VEL
LIN {X 0,Y 183.858,Z 385.317,A -85,B 0,C 180,E1 -22061.016,E2 -22061.016} C_VEL
LIN {X 0,Y 185.399,Z 382.159,A -85,B 0,C 180,E1 -22065.386,E2 -22065.386} C_VEL
LIN {X 0,Y 187.437,Z 378.682,A -85,B 0,C 180,E1 -22068.583,E2 -22068.583} C_VEL
LIN {X 0,Y 189.992,Z 374.182,A -85,B 0,C 180,E1 -22071.708,E2 -22071.708} C_VEL
LIN {X 0,Y 193.509,Z 367.525,A -85,B 0,C 180,E1 -22075.259,E2 -22075.259} C_VEL
LIN {X 0,Y 197.292,Z 360.355,A -85,B 0,C 180,E1 -22078.162,E2 -22078.162} C_VEL
LIN {X 0,Y 201.608,Z 351.563,A -85,B 0,C 180,E1 -22080.94,E2 -22080.94} C_VEL
LIN {X 0,Y 203.801,Z 342.903,A -85,B 0,C 180,E1 -22083.485,E2 -22083.485} C_VEL
LIN {X 0,Y 205.071,Z 333.551,A -85,B 0,C 180,E1 -22086.021,E2 -22086.021} C_VEL
LIN {X 0,Y 205.41,Z 324.572,A -85,B 0,C 180,E1 -22088.344,E2 -22088.344} C_VEL
LIN {X 0,Y 204.885,Z 314.02,A -85,B 0,C 180,E1 -22091.002,E2 -22091.002} C_VEL
LIN {X 0,Y 204.085,Z 308.551,A -85,B 0,C 180,E1 -22092.465,E2 -22092.465} C_VEL
LIN {X 0,Y 201.953,Z 302.557,A -85,B 0,C 180,E1 -22094.482,E2 -22094.482} C_VEL
LIN {X 0,Y 200.759,Z 299.546,A -85,B 0,C 180,E1 -22095.558,E2 -22095.558} C_VEL
LIN {X 0,Y 198.326,Z 294.263,A -85,B 0,C 180,E1 -22097.675,E2 -22097.675} C_VEL
LIN {X 0,Y 196.554,Z 291.39,A -85,B 0,C 180,E1 -22099.072,E2 -22099.072} C_VEL
LIN {X 0,Y 195.086,Z 288.066,A -85,B 0,C 180,E1 -22100.497,E2 -22100.497} C_VEL
LIN {X 0,Y 192.625,Z 284.224,A -85,B 0,C 180,E1 -22102.696,E2 -22102.696} C_VEL
LIN {X 0,Y 191.605,Z 281.699,A -85,B 0,C 180,E1 -22103.834,E2 -22103.834} C_VEL
LIN {X 0,Y 188.663,Z 278.165,A -85,B 0,C 180,E1 -22106.826,E2 -22106.826} C_VEL
LIN {X 0,Y 187.221,Z 274.839,A -85,B 0,C 180,E1 -22108.856,E2 -22108.856} C_VEL
LIN {X 0,Y 187.119,Z 274.339,A -85,B 0,C 180,E1 -22109.174,E2 -22109.174} C_VEL
LIN {X 0,Y 186.902,Z 272.438,A -85,B 0,C 180,E1 -22114.478,E2 -22114.478} C_VEL
LIN {X 0,Y 186.678,Z 270.946,A -85,B 0,C 180,E1 -22120.246,E2 -22120.246} C_VEL
LIN {X 0,Y 186.615,Z 270.221,A -85,B 0,C 180,E1 -22124.712,E2 -22124.712} C_VEL
LIN {X 0,Y 186.708,Z 269.727,A -85,B 0,C 180,E1 -22129.149,E2 -22129.149} C_VEL
LIN {X 0,Y 186.802,Z 269.621,A -85,B 0,C 180,E1 -22131.341,E2 -22131.341} C_VEL
LIN {X 0,Y 186.786,Z 269.726,A -85,B 0,C 180,E1 -22133.719,E2 -22133.719} C_VEL
LIN {X 0,Y 187.73,Z 271.909,A -85,B 0,C 180,E1 -22135.299,E2 -22135.299} C_VEL
LIN {X 0,Y 190.565,Z 274.352,A -85,B 0,C 180,E1 -22138.412,E2 -22138.412} C_VEL
LIN {X 0,Y 191.721,Z 275.099,A -85,B 0,C 180,E1 -22139.472,E2 -22139.472} C_VEL
LIN {X 0,Y 193.182,Z 278.143,A -85,B 0,C 180,E1 -22141.169,E2 -22141.169} C_VEL
LIN {X 0,Y 194.997,Z 279.97,A -85,B 0,C 180,E1 -22142.689,E2 -22142.689} C_VEL
LIN {X 0,Y 196.327,Z 282.89,A -85,B 0,C 180,E1 -22144.102,E2 -22144.102} C_VEL
LIN {X 0,Y 197.558,Z 284.407,A -85,B 0,C 180,E1 -22145.099,E2 -22145.099} C_VEL
LIN {X 0,Y 200.941,Z 290.346,A -85,B 0,C 180,E1 -22148.039,E2 -22148.039} C_VEL
LIN {X 0,Y 204.752,Z 298.945,A -85,B 0,C 180,E1 -22151.586,E2 -22151.586} C_VEL
LIN {X 0,Y 207.017,Z 306.265,A -85,B 0,C 180,E1 -22154.245,E2 -22154.245} C_VEL
LIN {X 0,Y 208.41,Z 314.403,A -85,B 0,C 180,E1 -22156.906,E2 -22156.906} C_VEL
LIN {X 0,Y 208.876,Z 321.515,A -85,B 0,C 180,E1 -22159.199,E2 -22159.199} C_VEL
LIN {X 0,Y 208.824,Z 324.551,A -85,B 0,C 180,E1 -22160.176,E2 -22160.176} C_VEL
LIN {X 0,Y 206.897,Z 329.627,A -85,B 0,C 180,E1 -22161.427,E2 -22161.427} C_VEL
LIN {X 0,Y 203.256,Z 337.453,A -85,B 0,C 180,E1 -22163.618,E2 -22163.618} C_VEL
LIN {X 0,Y 199.594,Z 344.599,A -85,B 0,C 180,E1 -22166.122,E2 -22166.122} C_VEL
LIN {X 0,Y 195.459,Z 351.797,A -85,B 0,C 180,E1 -22169.363,E2 -22169.363} C_VEL
LIN {X 0,Y 191.995,Z 357.321,A -85,B 0,C 180,E1 -22172.661,E2 -22172.661} C_VEL
LIN {X 0,Y 189.677,Z 360.779,A -85,B 0,C 180,E1 -22175.401,E2 -22175.401} C_VEL
LIN {X 0,Y 187.75,Z 363.451,A -85,B 0,C 180,E1 -22178.182,E2 -22178.182} C_VEL
LIN {X 0,Y 186.179,Z 365.38,A -85,B 0,C 180,E1 -22180.98,E2 -22180.98} C_VEL
LIN {X 0,Y 184.929,Z 366.574,A -85,B 0,C 180,E1 -22183.778,E2 -22183.778} C_VEL
LIN {X 0,Y 184.019,Z 367.149,A -85,B 0,C 180,E1 -22186.575,E2 -22186.575} C_VEL
LIN {X 0,Y 183.359,Z 366.96,A -85,B 0,C 180,E1 -22190.042,E2 -22190.042} C_VEL
LIN {X 0,Y 183.138,Z 365.704,A -85,B 0,C 180,E1 -22193.689,E2 -22193.689} C_VEL
LIN {X 0,Y 183.386,Z 363.159,A -85,B 0,C 180,E1 -22197.555,E2 -22197.555} C_VEL
LIN {X 0,Y 184.188,Z 359.363,A -85,B 0,C 180,E1 -22201.346,E2 -22201.346} C_VEL
LIN {X 0,Y 185.443,Z 353.644,A -85,B 0,C 180,E1 -22205.435,E2 -22205.435} C_VEL
LIN {X 0,Y 187.024,Z 347.326,A -85,B 0,C 180,E1 -22208.821,E2 -22208.821} C_VEL
LIN {X 0,Y 189.025,Z 339.461,A -85,B 0,C 180,E1 -22212.14,E2 -22212.14} C_VEL
LIN {X 0,Y 191.336,Z 330.535,A -85,B 0,C 180,E1 -22215.103,E2 -22215.103} C_VEL
LIN {X 0,Y 193.821,Z 320.365,A -85,B 0,C 180,E1 -22217.769,E2 -22217.769} C_VEL
LIN {X 0,Y 196.095,Z 309.979,A -85,B 0,C 180,E1 -22219.94,E2 -22219.94} C_VEL
LIN {X 0,Y 196.192,Z 307.318,A -85,B 0,C 180,E1 -22220.466,E2 -22220.466} C_VEL
LIN {X 0,Y 194.512,Z 296.47,A -85,B 0,C 180,E1 -22222.629,E2 -22222.629} C_VEL
LIN {X 0,Y 192.136,Z 285.3,A -85,B 0,C 180,E1 -22224.571,E2 -22224.571} C_VEL
LIN {X 0,Y 189.391,Z 275.413,A -85,B 0,C 180,E1 -22226.079,E2 -22226.079} C_VEL
LIN {X 0,Y 185.821,Z 266.137,A -85,B 0,C 180,E1 -22227.428,E2 -22227.428} C_VEL
LIN {X 0,Y 185.73,Z 265.348,A -85,B 0,C 180,E1 -22227.562,E2 -22227.562} C_VEL
LIN {X 0,Y 186.283,Z 265.28,A -85,B 0,C 180,E1 -22230.002,E2 -22230.002} C_VEL
LIN {X 0,Y 186.196,Z 265.292,A -85,B 0,C 180,E1 -22232.165,E2 -22232.165} C_VEL
LIN {X 0,Y 185.998,Z 265.312,A -85,B 0,C 180,E1 -22238.695,E2 -22238.695} C_VEL
LIN {X 0,Y 185.756,Z 265.344,A -85,B 0,C 180,E1 -22243.123,E2 -22243.123} C_VEL
LIN {X 0,Y 185.711,Z 265.356,A -85,B 0,C 180,E1 -22247.625,E2 -22247.625} C_VEL
LIN {X 0,Y 185.611,Z 265.356,A -85,B 0,C 180,E1 -22252.252,E2 -22252.252} C_VEL
LIN {X 0,Y 185.556,Z 265.376,A -85,B 0,C 180,E1 -22257.035,E2 -22257.035} C_VEL
LIN {X 0,Y 185.572,Z 265.372,A -85,B 0,C 180,E1 -22259.497,E2 -22259.497} C_VEL
LIN {X 0,Y 185.515,Z 265.376,A -85,B 0,C 180,E1 -22264.631,E2 -22264.631} C_VEL
LIN {X 0,Y 185.562,Z 265.371,A -85,B 0,C 180,E1 -22267.318,E2 -22267.318} C_VEL
LIN {X 0,Y 185.557,Z 265.372,A -85,B 0,C 180,E1 -22270.762,E2 -22270.762} C_VEL
LIN {X 0,Y 185.561,Z 265.366,A -85,B 0,C 180,E1 -22276.026,E2 -22276.026} C_VEL
LIN {X 0,Y 185.538,Z 265.373,A -85,B 0,C 180,E1 -22279.918,E2 -22279.918} C_VEL
LIN {X 0,Y 185.558,Z 265.36,A -85,B 0,C 180,E1 -22282.704,E2 -22282.704} C_VEL
LIN {X 0,Y 185.545,Z 265.36,A -85,B 0,C 180,E1 -22287.98,E2 -22287.98} C_VEL
LIN {X 0,Y 185.583,Z 265.367,A -85,B 0,C 180,E1 -22290.58,E2 -22290.58} C_VEL
LIN {X 0,Y 185.59,Z 265.362,A -85,B 0,C 180,E1 -22295.387,E2 -22295.387} C_VEL
LIN {X 0,Y 185.678,Z 265.338,A -85,B 0,C 180,E1 -22301.137,E2 -22301.137} C_VEL
LIN {X 0,Y 185.729,Z 265.346,A -85,B 0,C 180,E1 -22304.644,E2 -22304.644} C_VEL
LIN {X 0,Y 185.894,Z 265.327,A -85,B 0,C 180,E1 -22309.422,E2 -22309.422} C_VEL
LIN {X 0,Y 185.951,Z 265.302,A -85,B 0,C 180,E1 -22313.493,E2 -22313.493} C_VEL
LIN {X 0,Y 186.212,Z 265.283,A -85,B 0,C 180,E1 -22317.84,E2 -22317.84} C_VEL
LIN {X 0,Y 186.412,Z 265.265,A -85,B 0,C 180,E1 -22320.003,E2 -22320.003} C_VEL
LIN {X 0,Y 185.92,Z 265.319,A -85,B 0,C 180,E1 -22324.339,E2 -22324.339} C_VEL
LIN {X 0,Y 185.989,Z 265.303,A -85,B 0,C 180,E1 -22328.697,E2 -22328.697} C_VEL
LIN {X 0,Y 185.738,Z 265.349,A -85,B 0,C 180,E1 -22333.125,E2 -22333.125} C_VEL
LIN {X 0,Y 185.701,Z 265.343,A -85,B 0,C 180,E1 -22337.627,E2 -22337.627} C_VEL
LIN {X 0,Y 185.608,Z 265.364,A -85,B 0,C 180,E1 -22342.253,E2 -22342.253} C_VEL
LIN {X 0,Y 185.572,Z 265.362,A -85,B 0,C 180,E1 -22347.034,E2 -22347.034} C_VEL
LIN {X 0,Y 185.589,Z 265.365,A -85,B 0,C 180,E1 -22349.495,E2 -22349.495} C_VEL
LIN {X 0,Y 185.53,Z 265.374,A -85,B 0,C 180,E1 -22354.629,E2 -22354.629} C_VEL
LIN {X 0,Y 185.648,Z 265.596,A -85,B 0,C 180,E1 -22356.605,E2 -22356.605} C_VEL
LIN {X 0,Y 186.238,Z 268.865,A -85,B 0,C 180,E1 -22360.995,E2 -22360.995} C_VEL
LIN {X 0,Y 186.879,Z 272.504,A -85,B 0,C 180,E1 -22365.609,E2 -22365.609} C_VEL
LIN {X 0,Y 187.577,Z 276.539,A -85,B 0,C 180,E1 -22370.433,E2 -22370.433} C_VEL
LIN {X 0,Y 187.689,Z 277.789,A -85,B 0,C 180,E1 -22371.849,E2 -22371.849} C_VEL
LIN {X 0,Y 186.967,Z 281.093,A -85,B 0,C 180,E1 -22375.437,E2 -22375.437} C_VEL
LIN {X 0,Y 189.45,Z 295.389,A -85,B 0,C 180,E1 -22376.949,E2 -22376.949} C_VEL
LIN {X 0,Y 191.082,Z 307.812,A -85,B 0,C 180,E1 -22378.61,E2 -22378.61} C_VEL
LIN {X 0,Y 192.013,Z 319.67,A -85,B 0,C 180,E1 -22380.506,E2 -22380.506} C_VEL
LIN {X 0,Y 192.373,Z 330.301,A -85,B 0,C 180,E1 -22382.531,E2 -22382.531} C_VEL
LIN {X 0,Y 192.249,Z 340.535,A -85,B 0,C 180,E1 -22384.849,E2 -22384.849} C_VEL
LIN {X 0,Y 189.625,Z 351.274,A -85,B 0,C 180,E1 -22387.671,E2 -22387.671} C_VEL
LIN {X 0,Y 187.91,Z 358.143,A -85,B 0,C 180,E1 -22389.911,E2 -22389.911} C_VEL
LIN {X 0,Y 186.129,Z 365.84,A -85,B 0,C 180,E1 -22392.982,E2 -22392.982} C_VEL
LIN {X 0,Y 184.83,Z 371.312,A -85,B 0,C 180,E1 -22395.688,E2 -22395.688} C_VEL
LIN {X 0,Y 183.899,Z 376.667,A -85,B 0,C 180,E1 -22398.982,E2 -22398.982} C_VEL
LIN {X 0,Y 183.467,Z 380.815,A -85,B 0,C 180,E1 -22402.293,E2 -22402.293} C_VEL
LIN {X 0,Y 183.454,Z 383.868,A -85,B 0,C 180,E1 -22405.604,E2 -22405.604} C_VEL
LIN {X 0,Y 183.501,Z 385.352,A -85,B 0,C 180,E1 -22407.803,E2 -22407.803} C_VEL
LIN {X 0,Y 183.556,Z 386.362,A -85,B 0,C 180,E1 -22409.998,E2 -22409.998} C_VEL
LIN {X 0,Y 183.408,Z 386.942,A -85,B 0,C 180,E1 -22412.194,E2 -22412.194} C_VEL
LIN {X 0,Y 183.281,Z 386.929,A -85,B 0,C 180,E1 -22416.603,E2 -22416.603} C_VEL
LIN {X 0,Y 183.293,Z 386.832,A -85,B 0,C 180,E1 -22416.957,E2 -22416.957} C_VEL
LIN {X 0,Y 182.769,Z 386.317,A -85,B 0,C 180,E1 -22418.79,E2 -22418.79} C_VEL
LIN {X 0,Y 180.444,Z 384.88,A -85,B 0,C 180,E1 -22421.805,E2 -22421.805} C_VEL
LIN {X 0,Y 178.648,Z 382.932,A -85,B 0,C 180,E1 -22424.854,E2 -22424.854} C_VEL
LIN {X 0,Y 178.956,Z 381.384,A -85,B 0,C 180,E1 -22426.68,E2 -22426.68} C_VEL
LIN {X 0,Y 181.47,Z 377.316,A -85,B 0,C 180,E1 -22430.396,E2 -22430.396} C_VEL
LIN {X 0,Y 184.923,Z 371.558,A -85,B 0,C 180,E1 -22434.194,E2 -22434.194} C_VEL
LIN {X 0,Y 188.996,Z 364.475,A -85,B 0,C 180,E1 -22437.696,E2 -22437.696} C_VEL
LIN {X 0,Y 193.279,Z 356.711,A -85,B 0,C 180,E1 -22440.599,E2 -22440.599} C_VEL
LIN {X 0,Y 195.546,Z 352.182,A -85,B 0,C 180,E1 -22442.011,E2 -22442.011} C_VEL
LIN {X 0,Y 197.893,Z 343.794,A -85,B 0,C 180,E1 -22444.624,E2 -22444.624} C_VEL
LIN {X 0,Y 199.46,Z 333.481,A -85,B 0,C 180,E1 -22447.593,E2 -22447.593} C_VEL
LIN {X 0,Y 199.866,Z 323.078,A -85,B 0,C 180,E1 -22450.454,E2 -22450.454} C_VEL
LIN {X 0,Y 199.512,Z 315.145,A -85,B 0,C 180,E1 -22452.632,E2 -22452.632} C_VEL
LIN {X 0,Y 198.871,Z 311.301,A -85,B 0,C 180,E1 -22453.812,E2 -22453.812} C_VEL
LIN {X 0,Y 196.417,Z 304.333,A -85,B 0,C 180,E1 -22456.462,E2 -22456.462} C_VEL
LIN {X 0,Y 194.442,Z 299.609,A -85,B 0,C 180,E1 -22458.479,E2 -22458.479} C_VEL
LIN {X 0,Y 192.607,Z 295.804,A -85,B 0,C 180,E1 -22460.311,E2 -22460.311} C_VEL
LIN {X 0,Y 192.169,Z 294.464,A -85,B 0,C 180,E1 -22460.882,E2 -22460.882} C_VEL
LIN {X 0,Y 189.96,Z 290.929,A -85,B 0,C 180,E1 -22463.04,E2 -22463.04} C_VEL
LIN {X 0,Y 188.836,Z 287.919,A -85,B 0,C 180,E1 -22464.56,E2 -22464.56} C_VEL
LIN {X 0,Y 186.176,Z 284.265,A -85,B 0,C 180,E1 -22467.633,E2 -22467.633} C_VEL
LIN {X 0,Y 185.027,Z 280.93,A -85,B 0,C 180,E1 -22469.745,E2 -22469.745} C_VEL
LIN {X 0,Y 181.371,Z 276.293,A -85,B 0,C 180,E1 -22477.499,E2 -22477.499} C_VEL
LIN {X 0,Y 180.939,Z 274.898,A -85,B 0,C 180,E1 -22481.893,E2 -22481.893} C_VEL
LIN {X 0,Y 181.889,Z 275.111,A -85,B 0,C 180,E1 -22487.586,E2 -22487.586} C_VEL
LIN {X 0,Y 184.86,Z 276.639,A -85,B 0,C 180,E1 -22493.297,E2 -22493.297} C_VEL
LIN {X 0,Y 185.991,Z 279.034,A -85,B 0,C 180,E1 -22495.391,E2 -22495.391} C_VEL
LIN {X 0,Y 189.099,Z 281.611,A -85,B 0,C 180,E1 -22498.932,E2 -22498.932} C_VEL
LIN {X 0,Y 189.815,Z 283.472,A -85,B 0,C 180,E1 -22499.997,E2 -22499.997} C_VEL
LIN {X 0,Y 191.861,Z 286.126,A -85,B 0,C 180,E1 -22502.096,E2 -22502.096} C_VEL
LIN {X 0,Y 192.857,Z 288.533,A -85,B 0,C 180,E1 -22503.342,E2 -22503.342} C_VEL
LIN {X 0,Y 195.71,Z 293.327,A -85,B 0,C 180,E1 -22506.181,E2 -22506.181} C_VEL
LIN {X 0,Y 198.1,Z 298.547,A -85,B 0,C 180,E1 -22508.692,E2 -22508.692} C_VEL
LIN {X 0,Y 200.403,Z 304.826,A -85,B 0,C 180,E1 -22511.374,E2 -22511.374} C_VEL
LIN {X 0,Y 201.867,Z 310.573,A -85,B 0,C 180,E1 -22513.588,E2 -22513.588} C_VEL
LIN {X 0,Y 202.9,Z 319.129,A -85,B 0,C 180,E1 -22516.601,E2 -22516.601} C_VEL
LIN {X 0,Y 202.898,Z 326.823,A -85,B 0,C 180,E1 -22519.268,E2 -22519.268} C_VEL
LIN {X 0,Y 198.638,Z 336.043,A -85,B 0,C 180,E1 -22521.765,E2 -22521.765} C_VEL
LIN {X 0,Y 194.651,Z 343.568,A -85,B 0,C 180,E1 -22524.312,E2 -22524.312} C_VEL
LIN {X 0,Y 190.251,Z 351.018,A -85,B 0,C 180,E1 -22527.559,E2 -22527.559} C_VEL
LIN {X 0,Y 187.081,Z 355.792,A -85,B 0,C 180,E1 -22530.232,E2 -22530.232} C_VEL
LIN {X 0,Y 184.388,Z 359.642,A -85,B 0,C 180,E1 -22533.019,E2 -22533.019} C_VEL
LIN {X 0,Y 182.105,Z 362.669,A -85,B 0,C 180,E1 -22535.863,E2 -22535.863} C_VEL
LIN {X 0,Y 180.234,Z 364.952,A -85,B 0,C 180,E1 -22538.755,E2 -22538.755} C_VEL
LIN {X 0,Y 178.553,Z 366.64,A -85,B 0,C 180,E1 -22541.995,E2 -22541.995} C_VEL
LIN {X 0,Y 177.219,Z 367.523,A -85,B 0,C 180,E1 -22545.541,E2 -22545.541} C_VEL
LIN {X 0,Y 176.375,Z 367.436,A -85,B 0,C 180,E1 -22549.202,E2 -22549.202} C_VEL
LIN {X 0,Y 176.044,Z 366.201,A -85,B 0,C 180,E1 -22553.217,E2 -22553.217} C_VEL
LIN {X 0,Y 176.183,Z 363.988,A -85,B 0,C 180,E1 -22556.89,E2 -22556.89} C_VEL
LIN {X 0,Y 176.977,Z 360.308,A -85,B 0,C 180,E1 -22560.877,E2 -22560.877} C_VEL
LIN {X 0,Y 177.895,Z 356.085,A -85,B 0,C 180,E1 -22564.245,E2 -22564.245} C_VEL
LIN {X 0,Y 179.497,Z 349.63,A -85,B 0,C 180,E1 -22568.167,E2 -22568.167} C_VEL
LIN {X 0,Y 181.315,Z 342.902,A -85,B 0,C 180,E1 -22571.353,E2 -22571.353} C_VEL
LIN {X 0,Y 183.467,Z 334.693,A -85,B 0,C 180,E1 -22574.448,E2 -22574.448} C_VEL
LIN {X 0,Y 185.904,Z 325.459,A -85,B 0,C 180,E1 -22577.217,E2 -22577.217} C_VEL
LIN {X 0,Y 188.526,Z 314.611,A -85,B 0,C 180,E1 -22579.803,E2 -22579.803} C_VEL
LIN {X 0,Y 189.499,Z 309.025,A -85,B 0,C 180,E1 -22580.933,E2 -22580.933} C_VEL
LIN {X 0,Y 187.842,Z 297.889,A -85,B 0,C 180,E1 -22583.267,E2 -22583.267} C_VEL
LIN {X 0,Y 185.392,Z 286.14,A -85,B 0,C 180,E1 -22585.409,E2 -22585.409} C_VEL
LIN {X 0,Y 182.996,Z 277.499,A -85,B 0,C 180,E1 -22586.822,E2 -22586.822} C_VEL
LIN {X 0,Y 179.008,Z 267.167,A -85,B 0,C 180,E1 -22588.456,E2 -22588.456} C_VEL
LIN {X 0,Y 178.856,Z 266.204,A -85,B 0,C 180,E1 -22588.595,E2 -22588.595} C_VEL
LIN {X 0,Y 179.233,Z 266.158,A -85,B 0,C 180,E1 -22590.002,E2 -22590.002} C_VEL
LIN {X 0,Y 179.142,Z 266.171,A -85,B 0,C 180,E1 -22592.251,E2 -22592.251} C_VEL
LIN {X 0,Y 178.927,Z 266.192,A -85,B 0,C 180,E1 -22599.042,E2 -22599.042} C_VEL
LIN {X 0,Y 178.68,Z 266.223,A -85,B 0,C 180,E1 -22603.653,E2 -22603.653} C_VEL
LIN {X 0,Y 178.672,Z 266.233,A -85,B 0,C 180,E1 -22608.344,E2 -22608.344} C_VEL
LIN {X 0,Y 178.524,Z 266.244,A -85,B 0,C 180,E1 -22613.186,E2 -22613.186} C_VEL
LIN {X 0,Y 178.481,Z 266.255,A -85,B 0,C 180,E1 -22618.201,E2 -22618.201} C_VEL
LIN {X 0,Y 178.494,Z 266.256,A -85,B 0,C 180,E1 -22620.79,E2 -22620.79} C_VEL
LIN {X 0,Y 178.479,Z 266.251,A -85,B 0,C 180,E1 -22624.224,E2 -22624.224} C_VEL
LIN {X 0,Y 178.467,Z 266.251,A -85,B 0,C 180,E1 -22629.059,E2 -22629.059} C_VEL
LIN {X 0,Y 178.495,Z 266.251,A -85,B 0,C 180,E1 -22632.02,E2 -22632.02} C_VEL
LIN {X 0,Y 178.514,Z 266.243,A -85,B 0,C 180,E1 -22635.128,E2 -22635.128} C_VEL
LIN {X 0,Y 178.498,Z 266.252,A -85,B 0,C 180,E1 -22638.428,E2 -22638.428} C_VEL
LIN {X 0,Y 178.458,Z 266.239,A -85,B 0,C 180,E1 -22643.796,E2 -22643.796} C_VEL
LIN {X 0,Y 178.491,Z 266.23,A -85,B 0,C 180,E1 -22646.552,E2 -22646.552} C_VEL
LIN {X 0,Y 178.523,Z 266.242,A -85,B 0,C 180,E1 -22650.011,E2 -22650.011} C_VEL
LIN {X 0,Y 178.536,Z 266.241,A -85,B 0,C 180,E1 -22654.88,E2 -22654.88} C_VEL
LIN {X 0,Y 178.627,Z 266.213,A -85,B 0,C 180,E1 -22660.788,E2 -22660.788} C_VEL
LIN {X 0,Y 178.67,Z 266.222,A -85,B 0,C 180,E1 -22664.021,E2 -22664.021} C_VEL
LIN {X 0,Y 178.839,Z 266.205,A -85,B 0,C 180,E1 -22669.261,E2 -22669.261} C_VEL
LIN {X 0,Y 178.914,Z 266.179,A -85,B 0,C 180,E1 -22673.236,E2 -22673.236} C_VEL
LIN {X 0,Y 179.158,Z 266.16,A -85,B 0,C 180,E1 -22677.755,E2 -22677.755} C_VEL
LIN {X 0,Y 179.375,Z 266.142,A -85,B 0,C 180,E1 -22680.003,E2 -22680.003} C_VEL
LIN {X 0,Y 178.868,Z 266.197,A -85,B 0,C 180,E1 -22684.511,E2 -22684.511} C_VEL
LIN {X 0,Y 178.918,Z 266.184,A -85,B 0,C 180,E1 -22689.043,E2 -22689.043} C_VEL
LIN {X 0,Y 178.667,Z 266.231,A -85,B 0,C 180,E1 -22693.655,E2 -22693.655} C_VEL
LIN {X 0,Y 178.634,Z 266.22,A -85,B 0,C 180,E1 -22699.219,E2 -22699.219} C_VEL
LIN {X 0,Y 178.546,Z 266.244,A -85,B 0,C 180,E1 -22705.126,E2 -22705.126} C_VEL
LIN {X 0,Y 178.488,Z 266.251,A -85,B 0,C 180,E1 -22710.793,E2 -22710.793} C_VEL
LIN {X 0,Y 178.576,Z 266.449,A -85,B 0,C 180,E1 -22716.185,E2 -22716.185} C_VEL
LIN {X 0,Y 179.309,Z 270.542,A -85,B 0,C 180,E1 -22721.863,E2 -22721.863} C_VEL
LIN {X 0,Y 179.945,Z 274.061,A -85,B 0,C 180,E1 -22726.447,E2 -22726.447} C_VEL
LIN {X 0,Y 180.454,Z 276.869,A -85,B 0,C 180,E1 -22729.918,E2 -22729.918} C_VEL
LIN {X 0,Y 180.606,Z 278.186,A -85,B 0,C 180,E1 -22731.49,E2 -22731.49} C_VEL
LIN {X 0,Y 180.175,Z 280.702,A -85,B 0,C 180,E1 -22734.369,E2 -22734.369} C_VEL
LIN {X 0,Y 182.699,Z 295.234,A -85,B 0,C 180,E1 -22736.001,E2 -22736.001} C_VEL
LIN {X 0,Y 184.31,Z 307.663,A -85,B 0,C 180,E1 -22737.732,E2 -22737.732} C_VEL
LIN {X 0,Y 185.233,Z 320.162,A -85,B 0,C 180,E1 -22739.817,E2 -22739.817} C_VEL
LIN {X 0,Y 185.529,Z 331.4,A -85,B 0,C 180,E1 -22742.1,E2 -22742.1} C_VEL
LIN {X 0,Y 185.311,Z 341.141,A -85,B 0,C 180,E1 -22744.441,E2 -22744.441} C_VEL
LIN {X 0,Y 182.567,Z 351.702,A -85,B 0,C 180,E1 -22747.357,E2 -22747.357} C_VEL
LIN {X 0,Y 180.635,Z 359.528,A -85,B 0,C 180,E1 -22750.094,E2 -22750.094} C_VEL
LIN {X 0,Y 178.758,Z 367.155,A -85,B 0,C 180,E1 -22753.437,E2 -22753.437} C_VEL
LIN {X 0,Y 177.178,Z 374.173,A -85,B 0,C 180,E1 -22757.396,E2 -22757.396} C_VEL
LIN {X 0,Y 176.527,Z 378.816,A -85,B 0,C 180,E1 -22760.834,E2 -22760.834} C_VEL
LIN {X 0,Y 176.403,Z 382.838,A -85,B 0,C 180,E1 -22764.913,E2 -22764.913} C_VEL
LIN {X 0,Y 176.416,Z 384.759,A -85,B 0,C 180,E1 -22767.715,E2 -22767.715} C_VEL
LIN {X 0,Y 176.49,Z 385.851,A -85,B 0,C 180,E1 -22769.998,E2 -22769.998} C_VEL
LIN {X 0,Y 176.178,Z 386.691,A -85,B 0,C 180,E1 -22774.183,E2 -22774.183} C_VEL
LIN {X 0,Y 176.218,Z 386.521,A -85,B 0,C 180,E1 -22776.976,E2 -22776.976} C_VEL
LIN {X 0,Y 176.428,Z 386.015,A -85,B 0,C 180,E1 -22779.166,E2 -22779.166} C_VEL
LIN {X 0,Y 177.543,Z 383.734,A -85,B 0,C 180,E1 -22783.737,E2 -22783.737} C_VEL
LIN {X 0,Y 178.956,Z 381.384,A -85,B 0,C 180,E1 -22786.68,E2 -22786.68} C_VEL
LIN {X 0,Y 179.456,Z 379.678,A -85,B 0,C 180,E1 -22788.483,E2 -22788.483} C_VEL
LIN {X 0,Y 178.782,Z 376.501,A -85,B 0,C 180,E1 -22791.484,E2 -22791.484} C_VEL
LIN {X 0,Y 178.464,Z 372.72,A -85,B 0,C 180,E1 -22794.431,E2 -22794.431} C_VEL
LIN {X 0,Y 179.494,Z 370.049,A -85,B 0,C 180,E1 -22796.091,E2 -22796.091} C_VEL
LIN {X 0,Y 183.45,Z 363.655,A -85,B 0,C 180,E1 -22799.236,E2 -22799.236} C_VEL
LIN {X 0,Y 188.031,Z 355.832,A -85,B 0,C 180,E1 -22802.18,E2 -22802.18} C_VEL
LIN {X 0,Y 190.073,Z 351.334,A -85,B 0,C 180,E1 -22803.683,E2 -22803.683} C_VEL
LIN {X 0,Y 192.306,Z 343.578,A -85,B 0,C 180,E1 -22806.2,E2 -22806.2} C_VEL
LIN {X 0,Y 193.932,Z 333.632,A -85,B 0,C 180,E1 -22809.221,E2 -22809.221} C_VEL
LIN {X 0,Y 194.544,Z 323.344,A -85,B 0,C 180,E1 -22812.241,E2 -22812.241} C_VEL
LIN {X 0,Y 194.314,Z 317.209,A -85,B 0,C 180,E1 -22814.081,E2 -22814.081} C_VEL
LIN {X 0,Y 192.885,Z 311.831,A -85,B 0,C 180,E1 -22816.185,E2 -22816.185} C_VEL
LIN {X 0,Y 190.419,Z 304.899,A -85,B 0,C 180,E1 -22819.262,E2 -22819.262} C_VEL
LIN {X 0,Y 188.249,Z 299.605,A -85,B 0,C 180,E1 -22821.97,E2 -22821.97} C_VEL
LIN {X 0,Y 186.588,Z 296.442,A -85,B 0,C 180,E1 -22823.94,E2 -22823.94} C_VEL
LIN {X 0,Y 185.677,Z 293.87,A -85,B 0,C 180,E1 -22825.402,E2 -22825.402} C_VEL
LIN {X 0,Y 183.925,Z 291.32,A -85,B 0,C 180,E1 -22827.655,E2 -22827.655} C_VEL
LIN {X 0,Y 182.74,Z 288.078,A -85,B 0,C 180,E1 -22829.999,E2 -22829.999} C_VEL
LIN {X 0,Y 180.279,Z 284.393,A -85,B 0,C 180,E1 -22835.22,E2 -22835.22} C_VEL
LIN {X 0,Y 179.308,Z 282.198,A -85,B 0,C 180,E1 -22840.16,E2 -22840.16} C_VEL
LIN {X 0,Y 179.386,Z 281.682,A -85,B 0,C 180,E1 -22844.079,E2 -22844.079} C_VEL
LIN {X 0,Y 181.033,Z 282.501,A -85,B 0,C 180,E1 -22849.936,E2 -22849.936} C_VEL
LIN {X 0,Y 181.589,Z 282.753,A -85,B 0,C 180,E1 -22851.091,E2 -22851.091} C_VEL
LIN {X 0,Y 182.764,Z 283.97,A -85,B 0,C 180,E1 -22853.372,E2 -22853.372} C_VEL
LIN {X 0,Y 183.967,Z 286.106,A -85,B 0,C 180,E1 -22855.615,E2 -22855.615} C_VEL
LIN {X 0,Y 185.714,Z 287.553,A -85,B 0,C 180,E1 -22857.828,E2 -22857.828} C_VEL
LIN {X 0,Y 187.993,Z 291.472,A -85,B 0,C 180,E1 -22860.934,E2 -22860.934} C_VEL
LIN {X 0,Y 191.829,Z 299.007,A -85,B 0,C 180,E1 -22865.676,E2 -22865.676} C_VEL
LIN {X 0,Y 194.262,Z 305.367,A -85,B 0,C 180,E1 -22868.841,E2 -22868.841} C_VEL
LIN {X 0,Y 195.935,Z 310.958,A -85,B 0,C 180,E1 -22871.375,E2 -22871.375} C_VEL
LIN {X 0,Y 196.958,Z 317.448,A -85,B 0,C 180,E1 -22873.934,E2 -22873.934} C_VEL
LIN {X 0,Y 197.255,Z 324.362,A -85,B 0,C 180,E1 -22876.557,E2 -22876.557} C_VEL
LIN {X 0,Y 197.046,Z 328.736,A -85,B 0,C 180,E1 -22878.181,E2 -22878.181} C_VEL
LIN {X 0,Y 192.555,Z 337.888,A -85,B 0,C 180,E1 -22880.793,E2 -22880.793} C_VEL
LIN {X 0,Y 188.261,Z 345.37,A -85,B 0,C 180,E1 -22883.495,E2 -22883.495} C_VEL
LIN {X 0,Y 183.482,Z 352.755,A -85,B 0,C 180,E1 -22886.986,E2 -22886.986} C_VEL
LIN {X 0,Y 179.323,Z 358.503,A -85,B 0,C 180,E1 -22890.626,E2 -22890.626} C_VEL
LIN {X 0,Y 176.372,Z 362.263,A -85,B 0,C 180,E1 -22893.904,E2 -22893.904} C_VEL
LIN {X 0,Y 173.927,Z 365.047,A -85,B 0,C 180,E1 -22897.304,E2 -22897.304} C_VEL
LIN {X 0,Y 171.957,Z 366.919,A -85,B 0,C 180,E1 -22900.833,E2 -22900.833} C_VEL
LIN {X 0,Y 170.148,Z 367.991,A -85,B 0,C 180,E1 -22905.401,E2 -22905.401} C_VEL
LIN {X 0,Y 169.403,Z 367.884,A -85,B 0,C 180,E1 -22908.414,E2 -22908.414} C_VEL
LIN {X 0,Y 168.98,Z 366.878,A -85,B 0,C 180,E1 -22912.199,E2 -22912.199} C_VEL
LIN {X 0,Y 169.018,Z 364.699,A -85,B 0,C 180,E1 -22916.259,E2 -22916.259} C_VEL
LIN {X 0,Y 169.751,Z 361.224,A -85,B 0,C 180,E1 -22920.385,E2 -22920.385} C_VEL
LIN {X 0,Y 170.942,Z 355.957,A -85,B 0,C 180,E1 -22924.745,E2 -22924.745} C_VEL
LIN {X 0,Y 172.48,Z 349.956,A -85,B 0,C 180,E1 -22928.489,E2 -22928.489} C_VEL
LIN {X 0,Y 174.386,Z 343.198,A -85,B 0,C 180,E1 -22931.802,E2 -22931.802} C_VEL
LIN {X 0,Y 176.624,Z 334.957,A -85,B 0,C 180,E1 -22935.013,E2 -22935.013} C_VEL
LIN {X 0,Y 179.47,Z 324.484,A -85,B 0,C 180,E1 -22938.215,E2 -22938.215} C_VEL
LIN {X 0,Y 182.184,Z 313.399,A -85,B 0,C 180,E1 -22940.846,E2 -22940.846} C_VEL
LIN {X 0,Y 182.751,Z 310.591,A -85,B 0,C 180,E1 -22941.432,E2 -22941.432} C_VEL
LIN {X 0,Y 181.114,Z 299.029,A -85,B 0,C 180,E1 -22943.995,E2 -22943.995} C_VEL
LIN {X 0,Y 178.64,Z 286.857,A -85,B 0,C 180,E1 -22946.336,E2 -22946.336} C_VEL
LIN {X 0,Y 176.052,Z 278.415,A -85,B 0,C 180,E1 -22947.85,E2 -22947.85} C_VEL
LIN {X 0,Y 172.146,Z 267.625,A -85,B 0,C 180,E1 -22949.6,E2 -22949.6} C_VEL
LIN {X 0,Y 172.075,Z 267.051,A -85,B 0,C 180,E1 -22949.681,E2 -22949.681} C_VEL
LIN {X 0,Y 172.09,Z 267.049,A -85,B 0,C 180,E1 -22952.343,E2 -22952.343} C_VEL
LIN {X 0,Y 171.876,Z 267.077,A -85,B 0,C 180,E1 -22957.049,E2 -22957.049} C_VEL
LIN {X 0,Y 171.797,Z 267.085,A -85,B 0,C 180,E1 -22960.969,E2 -22960.969} C_VEL
LIN {X 0,Y 171.595,Z 267.112,A -85,B 0,C 180,E1 -22966.663,E2 -22966.663} C_VEL
LIN {X 0,Y 171.567,Z 267.115,A -85,B 0,C 180,E1 -22969.595,E2 -22969.595} C_VEL
LIN {X 0,Y 171.468,Z 267.131,A -85,B 0,C 180,E1 -22975.625,E2 -22975.625} C_VEL
LIN {X 0,Y 171.451,Z 267.132,A -85,B 0,C 180,E1 -22980.6,E2 -22980.6} C_VEL
LIN {X 0,Y 171.398,Z 267.137,A -85,B 0,C 180,E1 -22985.036,E2 -22985.036} C_VEL
LIN {X 0,Y 171.422,Z 267.129,A -85,B 0,C 180,E1 -22988.841,E2 -22988.841} C_VEL
LIN {X 0,Y 171.439,Z 267.129,A -85,B 0,C 180,E1 -22994.182,E2 -22994.182} C_VEL
LIN {X 0,Y 171.416,Z 267.132,A -85,B 0,C 180,E1 -22999.01,E2 -22999.01} C_VEL
LIN {X 0,Y 171.435,Z 267.123,A -85,B 0,C 180,E1 -23002.059,E2 -23002.059} C_VEL
LIN {X 0,Y 171.419,Z 267.118,A -85,B 0,C 180,E1 -23007.797,E2 -23007.797} C_VEL
LIN {X 0,Y 171.45,Z 267.126,A -85,B 0,C 180,E1 -23010.539,E2 -23010.539} C_VEL
LIN {X 0,Y 171.46,Z 267.121,A -85,B 0,C 180,E1 -23015.806,E2 -23015.806} C_VEL
LIN {X 0,Y 171.583,Z 267.09,A -85,B 0,C 180,E1 -23020.876,E2 -23020.876} C_VEL
LIN {X 0,Y 171.602,Z 267.107,A -85,B 0,C 180,E1 -23025.779,E2 -23025.779} C_VEL
LIN {X 0,Y 171.853,Z 267.07,A -85,B 0,C 180,E1 -23030.589,E2 -23030.589} C_VEL
LIN {X 0,Y 171.818,Z 267.061,A -85,B 0,C 180,E1 -23035.311,E2 -23035.311} C_VEL
LIN {X 0,Y 172.338,Z 267.018,A -85,B 0,C 180,E1 -23040.004,E2 -23040.004} C_VEL
LIN {X 0,Y 171.816,Z 267.076,A -85,B 0,C 180,E1 -23044.696,E2 -23044.696} C_VEL
LIN {X 0,Y 171.855,Z 267.065,A -85,B 0,C 180,E1 -23049.418,E2 -23049.418} C_VEL
LIN {X 0,Y 171.585,Z 267.111,A -85,B 0,C 180,E1 -23054.23,E2 -23054.23} C_VEL
LIN {X 0,Y 171.555,Z 267.103,A -85,B 0,C 180,E1 -23059.564,E2 -23059.564} C_VEL
LIN {X 0,Y 171.48,Z 267.121,A -85,B 0,C 180,E1 -23065.618,E2 -23065.618} C_VEL
LIN {X 0,Y 171.451,Z 267.127,A -85,B 0,C 180,E1 -23070.587,E2 -23070.587} C_VEL
LIN {X 0,Y 171.515,Z 267.277,A -85,B 0,C 180,E1 -23075.73,E2 -23075.73} C_VEL
LIN {X 0,Y 172.143,Z 270.758,A -85,B 0,C 180,E1 -23080.789,E2 -23080.789} C_VEL
LIN {X 0,Y 172.887,Z 274.78,A -85,B 0,C 180,E1 -23086.282,E2 -23086.282} C_VEL
LIN {X 0,Y 173.436,Z 277.956,A -85,B 0,C 180,E1 -23090.352,E2 -23090.352} C_VEL
LIN {X 0,Y 173.296,Z 280.405,A -85,B 0,C 180,E1 -23093.23,E2 -23093.23} C_VEL
LIN {X 0,Y 175.761,Z 293.626,A -85,B 0,C 180,E1 -23094.783,E2 -23094.783} C_VEL
LIN {X 0,Y 177.441,Z 306.148,A -85,B 0,C 180,E1 -23096.592,E2 -23096.592} C_VEL
LIN {X 0,Y 178.324,Z 318.017,A -85,B 0,C 180,E1 -23098.622,E2 -23098.622} C_VEL
LIN {X 0,Y 178.655,Z 329.098,A -85,B 0,C 180,E1 -23100.879,E2 -23100.879} C_VEL
LIN {X 0,Y 178.54,Z 339.47,A -85,B 0,C 180,E1 -23103.397,E2 -23103.397} C_VEL
LIN {X 0,Y 177.998,Z 342.726,A -85,B 0,C 180,E1 -23104.256,E2 -23104.256} C_VEL
LIN {X 0,Y 175.396,Z 352.477,A -85,B 0,C 180,E1 -23107.168,E2 -23107.168} C_VEL
LIN {X 0,Y 173.529,Z 359.722,A -85,B 0,C 180,E1 -23109.861,E2 -23109.861} C_VEL
LIN {X 0,Y 171.626,Z 367.234,A -85,B 0,C 180,E1 -23113.34,E2 -23113.34} C_VEL
LIN {X 0,Y 170.204,Z 373.248,A -85,B 0,C 180,E1 -23116.871,E2 -23116.871} C_VEL
LIN {X 0,Y 169.488,Z 377.999,A -85,B 0,C 180,E1 -23120.45,E2 -23120.45} C_VEL
LIN {X 0,Y 169.312,Z 380.544,A -85,B 0,C 180,E1 -23122.844,E2 -23122.844} C_VEL
LIN {X 0,Y 169.334,Z 382.568,A -85,B 0,C 180,E1 -23125.236,E2 -23125.236} C_VEL
LIN {X 0,Y 169.335,Z 384.143,A -85,B 0,C 180,E1 -23127.619,E2 -23127.619} C_VEL
LIN {X 0,Y 169.424,Z 385.299,A -85,B 0,C 180,E1 -23129.998,E2 -23129.998} C_VEL
LIN {X 0,Y 169.11,Z 386.247,A -85,B 0,C 180,E1 -23134.083,E2 -23134.083} C_VEL
LIN {X 0,Y 169.142,Z 386.162,A -85,B 0,C 180,E1 -23137.158,E2 -23137.158} C_VEL
LIN {X 0,Y 169.863,Z 384.818,A -85,B 0,C 180,E1 -23141.937,E2 -23141.937} C_VEL
LIN {X 0,Y 171.72,Z 381.883,A -85,B 0,C 180,E1 -23146.645,E2 -23146.645} C_VEL
LIN {X 0,Y 173.982,Z 378.632,A -85,B 0,C 180,E1 -23150.079,E2 -23150.079} C_VEL
LIN {X 0,Y 177.707,Z 373,A -85,B 0,C 180,E1 -23154.337,E2 -23154.337} C_VEL
LIN {X 0,Y 179.494,Z 370.049,A -85,B 0,C 180,E1 -23156.091,E2 -23156.091} C_VEL
LIN {X 0,Y 181.066,Z 366.259,A -85,B 0,C 180,E1 -23158.223,E2 -23158.223} C_VEL
LIN {X 0,Y 181.752,Z 362.322,A -85,B 0,C 180,E1 -23160.378,E2 -23160.378} C_VEL
LIN {X 0,Y 182.878,Z 355.797,A -85,B 0,C 180,E1 -23163.489,E2 -23163.489} C_VEL
LIN {X 0,Y 183.663,Z 353.375,A -85,B 0,C 180,E1 -23164.438,E2 -23164.438} C_VEL
LIN {X 0,Y 186.254,Z 345.642,A -85,B 0,C 180,E1 -23167.135,E2 -23167.135} C_VEL
LIN {X 0,Y 188.228,Z 336.24,A -85,B 0,C 180,E1 -23170.221,E2 -23170.221} C_VEL
LIN {X 0,Y 189.214,Z 326.649,A -85,B 0,C 180,E1 -23173.227,E2 -23173.227} C_VEL
LIN {X 0,Y 189.281,Z 320.829,A -85,B 0,C 180,E1 -23175.129,E2 -23175.129} C_VEL
LIN {X 0,Y 187.831,Z 314.944,A -85,B 0,C 180,E1 -23177.659,E2 -23177.659} C_VEL
LIN {X 0,Y 186.22,Z 310.022,A -85,B 0,C 180,E1 -23180.086,E2 -23180.086} C_VEL
LIN {X 0,Y 184.658,Z 305.487,A -85,B 0,C 180,E1 -23182.482,E2 -23182.482} C_VEL
LIN {X 0,Y 183.06,Z 301.888,A -85,B 0,C 180,E1 -23184.835,E2 -23184.835} C_VEL
LIN {X 0,Y 182.664,Z 300.35,A -85,B 0,C 180,E1 -23185.69,E2 -23185.69} C_VEL
LIN {X 0,Y 179.924,Z 294.268,A -85,B 0,C 180,E1 -23190.77,E2 -23190.77} C_VEL
LIN {X 0,Y 177.706,Z 290.449,A -85,B 0,C 180,E1 -23196.7,E2 -23196.7} C_VEL
LIN {X 0,Y 177.18,Z 288.688,A -85,B 0,C 180,E1 -23201.495,E2 -23201.495} C_VEL
LIN {X 0,Y 177.65,Z 288.616,A -85,B 0,C 180,E1 -23206.265,E2 -23206.265} C_VEL
LIN {X 0,Y 179.266,Z 289.464,A -85,B 0,C 180,E1 -23210.974,E2 -23210.974} C_VEL
LIN {X 0,Y 180.291,Z 290.767,A -85,B 0,C 180,E1 -23213.281,E2 -23213.281} C_VEL
LIN {X 0,Y 181.398,Z 292.726,A -85,B 0,C 180,E1 -23215.552,E2 -23215.552} C_VEL
LIN {X 0,Y 182.937,Z 294.265,A -85,B 0,C 180,E1 -23217.795,E2 -23217.795} C_VEL
LIN {X 0,Y 185.143,Z 298.779,A -85,B 0,C 180,E1 -23221.366,E2 -23221.366} C_VEL
LIN {X 0,Y 188.199,Z 305.622,A -85,B 0,C 180,E1 -23225.786,E2 -23225.786} C_VEL
LIN {X 0,Y 190.494,Z 313.521,A -85,B 0,C 180,E1 -23229.821,E2 -23229.821} C_VEL
LIN {X 0,Y 191.381,Z 318.784,A -85,B 0,C 180,E1 -23232.186,E2 -23232.186} C_VEL
LIN {X 0,Y 191.583,Z 325.354,A -85,B 0,C 180,E1 -23234.876,E2 -23234.876} C_VEL
LIN {X 0,Y 191.209,Z 330.965,A -85,B 0,C 180,E1 -23237.137,E2 -23237.137} C_VEL
LIN {X 0,Y 186.385,Z 339.862,A -85,B 0,C 180,E1 -23239.834,E2 -23239.834} C_VEL
LIN {X 0,Y 181.716,Z 347.402,A -85,B 0,C 180,E1 -23242.749,E2 -23242.749} C_VEL
LIN {X 0,Y 177.445,Z 353.557,A -85,B 0,C 180,E1 -23245.824,E2 -23245.824} C_VEL
LIN {X 0,Y 173.513,Z 358.566,A -85,B 0,C 180,E1 -23249.077,E2 -23249.077} C_VEL
LIN {X 0,Y 170.312,Z 362.385,A -85,B 0,C 180,E1 -23252.437,E2 -23252.437} C_VEL
LIN {X 0,Y 166.965,Z 365.872,A -85,B 0,C 180,E1 -23256.897,E2 -23256.897} C_VEL
LIN {X 0,Y 165.203,Z 367.387,A -85,B 0,C 180,E1 -23260.03,E2 -23260.03} C_VEL
LIN {X 0,Y 163.698,Z 368.257,A -85,B 0,C 180,E1 -23263.381,E2 -23263.381} C_VEL
LIN {X 0,Y 162.558,Z 368.357,A -85,B 0,C 180,E1 -23267.299,E2 -23267.299} C_VEL
LIN {X 0,Y 161.948,Z 367.441,A -85,B 0,C 180,E1 -23271.358,E2 -23271.358} C_VEL
LIN {X 0,Y 161.888,Z 365.341,A -85,B 0,C 180,E1 -23275.645,E2 -23275.645} C_VEL
LIN {X 0,Y 162.508,Z 362.065,A -85,B 0,C 180,E1 -23279.867,E2 -23279.867} C_VEL
LIN {X 0,Y 163.671,Z 357.057,A -85,B 0,C 180,E1 -23284.377,E2 -23284.377} C_VEL
LIN {X 0,Y 165.232,Z 351.141,A -85,B 0,C 180,E1 -23288.333,E2 -23288.333} C_VEL
LIN {X 0,Y 167.433,Z 343.506,A -85,B 0,C 180,E1 -23292.285,E2 -23292.285} C_VEL
LIN {X 0,Y 169.769,Z 335.235,A -85,B 0,C 180,E1 -23295.621,E2 -23295.621} C_VEL
LIN {X 0,Y 172.183,Z 326.662,A -85,B 0,C 180,E1 -23298.388,E2 -23298.388} C_VEL
LIN {X 0,Y 174.895,Z 316.374,A -85,B 0,C 180,E1 -23301.044,E2 -23301.044} C_VEL
LIN {X 0,Y 175.915,Z 312.155,A -85,B 0,C 180,E1 -23301.964,E2 -23301.964} C_VEL
LIN {X 0,Y 174.793,Z 302.621,A -85,B 0,C 180,E1 -23304.233,E2 -23304.233} C_VEL
LIN {X 0,Y 172.714,Z 291.232,A -85,B 0,C 180,E1 -23306.632,E2 -23306.632} C_VEL
LIN {X 0,Y 170.937,Z 284.196,A -85,B 0,C 180,E1 -23307.97,E2 -23307.97} C_VEL
LIN {X 0,Y 166.147,Z 270.849,A -85,B 0,C 180,E1 -23310.419,E2 -23310.419} C_VEL
LIN {X 0,Y 165.069,Z 267.92,A -85,B 0,C 180,E1 -23310.917,E2 -23310.917} C_VEL
LIN {X 0,Y 164.761,Z 267.958,A -85,B 0,C 180,E1 -23314.896,E2 -23314.896} C_VEL
LIN {X 0,Y 164.836,Z 267.952,A -85,B 0,C 180,E1 -23317.351,E2 -23317.351} C_VEL
LIN {X 0,Y 164.74,Z 267.965,A -85,B 0,C 180,E1 -23321.149,E2 -23321.149} C_VEL
LIN {X 0,Y 164.519,Z 267.997,A -85,B 0,C 180,E1 -23327.402,E2 -23327.402} C_VEL
LIN {X 0,Y 164.511,Z 267.994,A -85,B 0,C 180,E1 -23329.987,E2 -23329.987} C_VEL
LIN {X 0,Y 164.391,Z 268.013,A -85,B 0,C 180,E1 -23336.142,E2 -23336.142} C_VEL
LIN {X 0,Y 164.382,Z 268.013,A -85,B 0,C 180,E1 -23341.24,E2 -23341.24} C_VEL
LIN {X 0,Y 164.342,Z 268.017,A -85,B 0,C 180,E1 -23346.78,E2 -23346.78} C_VEL
LIN {X 0,Y 164.364,Z 268.007,A -85,B 0,C 180,E1 -23349.898,E2 -23349.898} C_VEL
LIN {X 0,Y 164.375,Z 268.008,A -85,B 0,C 180,E1 -23353.383,E2 -23353.383} C_VEL
LIN {X 0,Y 164.381,Z 268.008,A -85,B 0,C 180,E1 -23356.843,E2 -23356.843} C_VEL
LIN {X 0,Y 164.368,Z 268.009,A -85,B 0,C 180,E1 -23360.325,E2 -23360.325} C_VEL
LIN {X 0,Y 164.343,Z 267.99,A -85,B 0,C 180,E1 -23364.347,E2 -23364.347} C_VEL
LIN {X 0,Y 164.391,Z 268.001,A -85,B 0,C 180,E1 -23369.14,E2 -23369.14} C_VEL
LIN {X 0,Y 164.418,Z 268,A -85,B 0,C 180,E1 -23374.699,E2 -23374.699} C_VEL
LIN {X 0,Y 164.488,Z 267.969,A -85,B 0,C 180,E1 -23380.056,E2 -23380.056} C_VEL
LIN {X 0,Y 164.55,Z 267.984,A -85,B 0,C 180,E1 -23385.156,E2 -23385.156} C_VEL
LIN {X 0,Y 164.773,Z 267.953,A -85,B 0,C 180,E1 -23390.181,E2 -23390.181} C_VEL
LIN {X 0,Y 164.835,Z 267.934,A -85,B 0,C 180,E1 -23392.655,E2 -23392.655} C_VEL
LIN {X 0,Y 165.053,Z 267.915,A -85,B 0,C 180,E1 -23397.563,E2 -23397.563} C_VEL
LIN {X 0,Y 165.301,Z 267.895,A -85,B 0,C 180,E1 -23400.004,E2 -23400.004} C_VEL
LIN {X 0,Y 164.765,Z 267.954,A -85,B 0,C 180,E1 -23404.898,E2 -23404.898} C_VEL
LIN {X 0,Y 164.836,Z 267.932,A -85,B 0,C 180,E1 -23407.353,E2 -23407.353} C_VEL
LIN {X 0,Y 164.712,Z 267.963,A -85,B 0,C 180,E1 -23411.064,E2 -23411.064} C_VEL
LIN {X 0,Y 164.494,Z 267.984,A -85,B 0,C 180,E1 -23417.406,E2 -23417.406} C_VEL
LIN {X 0,Y 164.484,Z 267.986,A -85,B 0,C 180,E1 -23419.992,E2 -23419.992} C_VEL
LIN {X 0,Y 164.404,Z 268.001,A -85,B 0,C 180,E1 -23426.135,E2 -23426.135} C_VEL
LIN {X 0,Y 164.385,Z 268.01,A -85,B 0,C 180,E1 -23431.229,E2 -23431.229} C_VEL
LIN {X 0,Y 164.441,Z 268.034,A -85,B 0,C 180,E1 -23435.127,E2 -23435.127} C_VEL
LIN {X 0,Y 165.151,Z 272.076,A -85,B 0,C 180,E1 -23441.272,E2 -23441.272} C_VEL
LIN {X 0,Y 165.805,Z 275.498,A -85,B 0,C 180,E1 -23446.107,E2 -23446.107} C_VEL
LIN {X 0,Y 166.345,Z 278.937,A -85,B 0,C 180,E1 -23450.67,E2 -23450.67} C_VEL
LIN {X 0,Y 166.343,Z 279.913,A -85,B 0,C 180,E1 -23451.921,E2 -23451.921} C_VEL
LIN {X 0,Y 168.74,Z 291.378,A -85,B 0,C 180,E1 -23453.406,E2 -23453.406} C_VEL
LIN {X 0,Y 170.473,Z 304.156,A -85,B 0,C 180,E1 -23455.261,E2 -23455.261} C_VEL
LIN {X 0,Y 171.459,Z 315.989,A -85,B 0,C 180,E1 -23457.349,E2 -23457.349} C_VEL
LIN {X 0,Y 171.826,Z 328.008,A -85,B 0,C 180,E1 -23459.867,E2 -23459.867} C_VEL
LIN {X 0,Y 171.626,Z 338.799,A -85,B 0,C 180,E1 -23462.566,E2 -23462.566} C_VEL
LIN {X 0,Y 171.304,Z 342.126,A -85,B 0,C 180,E1 -23463.5,E2 -23463.5} C_VEL
LIN {X 0,Y 168.616,Z 351.86,A -85,B 0,C 180,E1 -23466.494,E2 -23466.494} C_VEL
LIN {X 0,Y 166.422,Z 359.867,A -85,B 0,C 180,E1 -23469.608,E2 -23469.608} C_VEL
LIN {X 0,Y 164.484,Z 367.283,A -85,B 0,C 180,E1 -23473.235,E2 -23473.235} C_VEL
LIN {X 0,Y 162.937,Z 374.084,A -85,B 0,C 180,E1 -23477.543,E2 -23477.543} C_VEL
LIN {X 0,Y 162.318,Z 378.548,A -85,B 0,C 180,E1 -23481.281,E2 -23481.281} C_VEL
LIN {X 0,Y 162.263,Z 381.903,A -85,B 0,C 180,E1 -23485.028,E2 -23485.028} C_VEL
LIN {X 0,Y 162.256,Z 383.527,A -85,B 0,C 180,E1 -23487.515,E2 -23487.515} C_VEL
LIN {X 0,Y 162.359,Z 384.732,A -85,B 0,C 180,E1 -23489.997,E2 -23489.997} C_VEL
LIN {X 0,Y 162.051,Z 385.741,A -85,B 0,C 180,E1 -23494.02,E2 -23494.02} C_VEL
LIN {X 0,Y 162.076,Z 385.779,A -85,B 0,C 180,E1 -23497.472,E2 -23497.472} C_VEL
LIN {X 0,Y 162.874,Z 384.542,A -85,B 0,C 180,E1 -23502.457,E2 -23502.457} C_VEL
LIN {X 0,Y 163.695,Z 383.363,A -85,B 0,C 180,E1 -23504.925,E2 -23504.925} C_VEL
LIN {X 0,Y 166.457,Z 379.758,A -85,B 0,C 180,E1 -23509.738,E2 -23509.738} C_VEL
LIN {X 0,Y 169.261,Z 375.96,A -85,B 0,C 180,E1 -23513.229,E2 -23513.229} C_VEL
LIN {X 0,Y 172.96,Z 370.557,A -85,B 0,C 180,E1 -23516.965,E2 -23516.965} C_VEL
LIN {X 0,Y 177.297,Z 364.046,A -85,B 0,C 180,E1 -23520.356,E2 -23520.356} C_VEL
LIN {X 0,Y 182.097,Z 356.453,A -85,B 0,C 180,E1 -23523.363,E2 -23523.363} C_VEL
LIN {X 0,Y 183.663,Z 353.375,A -85,B 0,C 180,E1 -23524.438,E2 -23524.438} C_VEL
LIN {X 0,Y 184.423,Z 349.812,A -85,B 0,C 180,E1 -23525.883,E2 -23525.883} C_VEL
LIN {X 0,Y 184.243,Z 346.523,A -85,B 0,C 180,E1 -23527.423,E2 -23527.423} C_VEL
LIN {X 0,Y 183.047,Z 340.037,A -85,B 0,C 180,E1 -23530.571,E2 -23530.571} C_VEL
LIN {X 0,Y 182.982,Z 336.382,A -85,B 0,C 180,E1 -23532.067,E2 -23532.067} C_VEL
LIN {X 0,Y 183.154,Z 335.05,A -85,B 0,C 180,E1 -23532.533,E2 -23532.533} C_VEL
LIN {X 0,Y 184.064,Z 327.763,A -85,B 0,C 180,E1 -23534.991,E2 -23534.991} C_VEL
LIN {X 0,Y 184.203,Z 325.285,A -85,B 0,C 180,E1 -23535.866,E2 -23535.866} C_VEL
LIN {X 0,Y 183.473,Z 321.188,A -85,B 0,C 180,E1 -23537.697,E2 -23537.697} C_VEL
LIN {X 0,Y 182.08,Z 315.659,A -85,B 0,C 180,E1 -23540.527,E2 -23540.527} C_VEL
LIN {X 0,Y 180.546,Z 310.704,A -85,B 0,C 180,E1 -23543.39,E2 -23543.39} C_VEL
LIN {X 0,Y 178.946,Z 305.84,A -85,B 0,C 180,E1 -23546.64,E2 -23546.64} C_VEL
LIN {X 0,Y 176.86,Z 300.333,A -85,B 0,C 180,E1 -23551.516,E2 -23551.516} C_VEL
LIN {X 0,Y 175.035,Z 296.796,A -85,B 0,C 180,E1 -23557.436,E2 -23557.436} C_VEL
LIN {X 0,Y 174.762,Z 295.445,A -85,B 0,C 180,E1 -23561.23,E2 -23561.23} C_VEL
LIN {X 0,Y 175.127,Z 295.239,A -85,B 0,C 180,E1 -23566.064,E2 -23566.064} C_VEL
LIN {X 0,Y 176.605,Z 296.022,A -85,B 0,C 180,E1 -23570.837,E2 -23570.837} C_VEL
LIN {X 0,Y 177.492,Z 297.348,A -85,B 0,C 180,E1 -23573.174,E2 -23573.174} C_VEL
LIN {X 0,Y 179.795,Z 300.835,A -85,B 0,C 180,E1 -23577.756,E2 -23577.756} C_VEL
LIN {X 0,Y 181.242,Z 304.188,A -85,B 0,C 180,E1 -23580.573,E2 -23580.573} C_VEL
LIN {X 0,Y 183.334,Z 309.609,A -85,B 0,C 180,E1 -23584.394,E2 -23584.394} C_VEL
LIN {X 0,Y 184.865,Z 315.201,A -85,B 0,C 180,E1 -23587.643,E2 -23587.643} C_VEL
LIN {X 0,Y 185.869,Z 320.868,A -85,B 0,C 180,E1 -23590.56,E2 -23590.56} C_VEL
LIN {X 0,Y 185.972,Z 327.746,A -85,B 0,C 180,E1 -23593.658,E2 -23593.658} C_VEL
LIN {X 0,Y 185.314,Z 333.404,A -85,B 0,C 180,E1 -23596.103,E2 -23596.103} C_VEL
LIN {X 0,Y 179.991,Z 342.387,A -85,B 0,C 180,E1 -23598.999,E2 -23598.999} C_VEL
LIN {X 0,Y 174.686,Z 350.094,A -85,B 0,C 180,E1 -23602.286,E2 -23602.286} C_VEL
LIN {X 0,Y 170.747,Z 355.24,A -85,B 0,C 180,E1 -23605.111,E2 -23605.111} C_VEL
LIN {X 0,Y 167.187,Z 359.439,A -85,B 0,C 180,E1 -23608.027,E2 -23608.027} C_VEL
LIN {X 0,Y 162.791,Z 364.147,A -85,B 0,C 180,E1 -23612.669,E2 -23612.669} C_VEL
LIN {X 0,Y 159.403,Z 367.198,A -85,B 0,C 180,E1 -23617.48,E2 -23617.48} C_VEL
LIN {X 0,Y 157.024,Z 368.628,A -85,B 0,C 180,E1 -23622.166,E2 -23622.166} C_VEL
LIN {X 0,Y 155.449,Z 368.707,A -85,B 0,C 180,E1 -23627.303,E2 -23627.303} C_VEL
LIN {X 0,Y 154.905,Z 367.958,A -85,B 0,C 180,E1 -23630.57,E2 -23630.57} C_VEL
LIN {X 0,Y 154.761,Z 366.062,A -85,B 0,C 180,E1 -23634.819,E2 -23634.819} C_VEL
LIN {X 0,Y 155.304,Z 362.877,A -85,B 0,C 180,E1 -23639.286,E2 -23639.286} C_VEL
LIN {X 0,Y 156.42,Z 358.104,A -85,B 0,C 180,E1 -23643.964,E2 -23643.964} C_VEL
LIN {X 0,Y 157.74,Z 353.096,A -85,B 0,C 180,E1 -23647.647,E2 -23647.647} C_VEL
LIN {X 0,Y 159.615,Z 346.646,A -85,B 0,C 180,E1 -23651.387,E2 -23651.387} C_VEL
LIN {X 0,Y 161.935,Z 338.959,A -85,B 0,C 180,E1 -23654.909,E2 -23654.909} C_VEL
